LIN {X 0,Y 239.969,Z 223.755,A -85,B 0,C 180,E1 -22346.527,E2 -22346.527} C_VEL
LIN {X 0,Y 242.861,Z 228.839,A -85,B 0,C 180,E1 -22348.912,E2 -22348.912} C_VEL
LIN {X 0,Y 246.024,Z 234.682,A -85,B 0,C 180,E1 -22351.164,E2 -22351.164} C_VEL
LIN {X 0,Y 248.847,Z 240.046,A -85,B 0,C 180,E1 -22352.983,E2 -22352.983} C_VEL
LIN {X 0,Y 253.177,Z 249.294,A -85,B 0,C 180,E1 -22355.55,E2 -22355.55} C_VEL
LIN {X 0,Y 256.52,Z 257.154,A -85,B 0,C 180,E1 -22357.368,E2 -22357.368} C_VEL
LIN {X 0,Y 257.027,Z 259.364,A -85,B 0,C 180,E1 -22357.681,E2 -22357.681} C_VEL
LIN {X 0,Y 256.983,Z 262.913,A -85,B 0,C 180,E1 -22357.859,E2 -22357.859} C_VEL
LIN {X 0,Y 256.14,Z 267.671,A -85,B 0,C 180,E1 -22357.804,E2 -22357.804} C_VEL
LIN {X 0,Y 255.103,Z 271.378,A -85,B 0,C 180,E1 -22357.618,E2 -22357.618} C_VEL
LIN {X 0,Y 251.834,Z 281.658,A -85,B 0,C 180,E1 -22356.935,E2 -22356.935} C_VEL
LIN {X 0,Y 250.756,Z 287.02,A -85,B 0,C 180,E1 -22356.819,E2 -22356.819} C_VEL
LIN {X 0,Y 250.638,Z 288.109,A -85,B 0,C 180,E1 -22356.836,E2 -22356.836} C_VEL
LIN {X 0,Y 247.434,Z 325.09,A -85,B 0,C 180,E1 -22357.818,E2 -22357.818} C_VEL
LIN {X 0,Y 244.93,Z 340.568,A -85,B 0,C 180,E1 -22358.4,E2 -22358.4} C_VEL
LIN {X 0,Y 241.457,Z 355.534,A -85,B 0,C 180,E1 -22359.199,E2 -22359.199} C_VEL
LIN {X 0,Y 237.664,Z 368.105,A -85,B 0,C 180,E1 -22360.08,E2 -22360.08} C_VEL
LIN {X 0,Y 232.84,Z 381.625,A -85,B 0,C 180,E1 -22361.339,E2 -22361.339} C_VEL
LIN {X 0,Y 227.303,Z 394.667,A -85,B 0,C 180,E1 -22362.894,E2 -22362.894} C_VEL
LIN {X 0,Y 221.538,Z 406.76,A -85,B 0,C 180,E1 -22364.781,E2 -22364.781} C_VEL
LIN {X 0,Y 216.696,Z 415.667,A -85,B 0,C 180,E1 -22366.435,E2 -22366.435} C_VEL
LIN {X 0,Y 210.539,Z 425.809,A -85,B 0,C 180,E1 -22368.756,E2 -22368.756} C_VEL
LIN {X 0,Y 203.927,Z 435.781,A -85,B 0,C 180,E1 -22371.66,E2 -22371.66} C_VEL
LIN {X 0,Y 197.461,Z 444.613,A -85,B 0,C 180,E1 -22374.945,E2 -22374.945} C_VEL
LIN {X 0,Y 192.716,Z 451.07,A -85,B 0,C 180,E1 -22378.077,E2 -22378.077} C_VEL
LIN {X 0,Y 187.417,Z 457.586,A -85,B 0,C 180,E1 -22382.048,E2 -22382.048} C_VEL
LIN {X 0,Y 183.132,Z 462.73,A -85,B 0,C 180,E1 -22386.238,E2 -22386.238} C_VEL
LIN {X 0,Y 180.543,Z 465.734,A -85,B 0,C 180,E1 -22389.493,E2 -22389.493} C_VEL
LIN {X 0,Y 178.115,Z 468.722,A -85,B 0,C 180,E1 -22393.967,E2 -22393.967} C_VEL
LIN {X 0,Y 176.609,Z 470.59,A -85,B 0,C 180,E1 -22398.524,E2 -22398.524} C_VEL
LIN {X 0,Y 175.965,Z 471.317,A -85,B 0,C 180,E1 -22403.119,E2 -22403.119} C_VEL
LIN {X 0,Y 175.967,Z 470.901,A -85,B 0,C 180,E1 -22407.712,E2 -22407.712} C_VEL
LIN {X 0,Y 176.119,Z 470.269,A -85,B 0,C 180,E1 -22410.001,E2 -22410.001} C_VEL
LIN {X 0,Y 176.018,Z 468.093,A -85,B 0,C 180,E1 -22414.581,E2 -22414.581} C_VEL
LIN {X 0,Y 176.233,Z 464.666,A -85,B 0,C 180,E1 -22419.18,E2 -22419.18} C_VEL
LIN {X 0,Y 177.037,Z 459.891,A -85,B 0,C 180,E1 -22423.781,E2 -22423.781} C_VEL
LIN {X 0,Y 178.755,Z 453.644,A -85,B 0,C 180,E1 -22428.334,E2 -22428.334} C_VEL
LIN {X 0,Y 181.359,Z 445.739,A -85,B 0,C 180,E1 -22432.801,E2 -22432.801} C_VEL
LIN {X 0,Y 184.466,Z 437.297,A -85,B 0,C 180,E1 -22436.595,E2 -22436.595} C_VEL
LIN {X 0,Y 188.286,Z 427.088,A -85,B 0,C 180,E1 -22440.26,E2 -22440.26} C_VEL
LIN {X 0,Y 192.055,Z 416.618,A -85,B 0,C 180,E1 -22443.293,E2 -22443.293} C_VEL
LIN {X 0,Y 196.36,Z 404.072,A -85,B 0,C 180,E1 -22446.198,E2 -22446.198} C_VEL
LIN {X 0,Y 199.968,Z 392.825,A -85,B 0,C 180,E1 -22448.277,E2 -22448.277} C_VEL
LIN {X 0,Y 203.401,Z 380.951,A -85,B 0,C 180,E1 -22450.057,E2 -22450.057} C_VEL
LIN {X 0,Y 206.679,Z 367.637,A -85,B 0,C 180,E1 -22451.668,E2 -22451.668} C_VEL
LIN {X 0,Y 209.533,Z 353.912,A -85,B 0,C 180,E1 -22452.947,E2 -22452.947} C_VEL
LIN {X 0,Y 211.958,Z 339.018,A -85,B 0,C 180,E1 -22453.968,E2 -22453.968} C_VEL
LIN {X 0,Y 213.625,Z 323.778,A -85,B 0,C 180,E1 -22454.686,E2 -22454.686} C_VEL
LIN {X 0,Y 218.933,Z 239.212,A -85,B 0,C 180,E1 -22457.242,E2 -22457.242} C_VEL
LIN {X 0,Y 218.792,Z 237.497,A -85,B 0,C 180,E1 -22457.347,E2 -22457.347} C_VEL
LIN {X 0,Y 212.348,Z 220.9,A -85,B 0,C 180,E1 -22459.583,E2 -22459.583} C_VEL
LIN {X 0,Y 206.415,Z 207.779,A -85,B 0,C 180,E1 -22461.739,E2 -22461.739} C_VEL
LIN {X 0,Y 200.574,Z 196.158,A -85,B 0,C 180,E1 -22464.009,E2 -22464.009} C_VEL
LIN {X 0,Y 196.878,Z 189.859,A -85,B 0,C 180,E1 -22465.51,E2 -22465.51} C_VEL
LIN {X 0,Y 191.655,Z 182.342,A -85,B 0,C 180,E1 -22467.702,E2 -22467.702} C_VEL
LIN {X 0,Y 188.625,Z 178.111,A -85,B 0,C 180,E1 -22469.066,E2 -22469.066} C_VEL
LIN {X 0,Y 185.755,Z 174.12,A -85,B 0,C 180,E1 -22470.429,E2 -22470.429} C_VEL
LIN {X 0,Y 183.259,Z 171.243,A -85,B 0,C 180,E1 -22471.647,E2 -22471.647} C_VEL
LIN {X 0,Y 182.122,Z 169.152,A -85,B 0,C 180,E1 -22472.278,E2 -22472.278} C_VEL
LIN {X 0,Y 179.819,Z 167.216,A -85,B 0,C 180,E1 -22473.448,E2 -22473.448} C_VEL
LIN {X 0,Y 178.609,Z 164.655,A -85,B 0,C 180,E1 -22474.197,E2 -22474.197} C_VEL
LIN {X 0,Y 178.489,Z 163.848,A -85,B 0,C 180,E1 -22474.335,E2 -22474.335} C_VEL
LIN {X 0,Y 178.521,Z 163.862,A -85,B 0,C 180,E1 -22479.25,E2 -22479.25} C_VEL
LIN {X 0,Y 178.649,Z 163.849,A -85,B 0,C 180,E1 -22481.657,E2 -22481.657} C_VEL
LIN {X 0,Y 178.653,Z 163.852,A -85,B 0,C 180,E1 -22486.348,E2 -22486.348} C_VEL
LIN {X 0,Y 178.908,Z 163.82,A -85,B 0,C 180,E1 -22490.961,E2 -22490.961} C_VEL
LIN {X 0,Y 179.128,Z 163.756,A -85,B 0,C 180,E1 -22497.752,E2 -22497.752} C_VEL
LIN {X 0,Y 179.348,Z 163.718,A -85,B 0,C 180,E1 -22500.001,E2 -22500.001} C_VEL
LIN {X 0,Y 178.834,Z 163.832,A -85,B 0,C 180,E1 -22504.509,E2 -22504.509} C_VEL
LIN {X 0,Y 178.907,Z 163.771,A -85,B 0,C 180,E1 -22509.041,E2 -22509.041} C_VEL
LIN {X 0,Y 178.633,Z 163.853,A -85,B 0,C 180,E1 -22513.655,E2 -22513.655} C_VEL
LIN {X 0,Y 178.558,Z 163.866,A -85,B 0,C 180,E1 -22519.151,E2 -22519.151} C_VEL
LIN {X 0,Y 178.509,Z 163.873,A -85,B 0,C 180,E1 -22525.104,E2 -22525.104} C_VEL
LIN {X 0,Y 178.465,Z 163.836,A -85,B 0,C 180,E1 -22530.795,E2 -22530.795} C_VEL
LIN {X 0,Y 178.487,Z 163.876,A -85,B 0,C 180,E1 -22534.218,E2 -22534.218} C_VEL
LIN {X 0,Y 178.392,Z 163.849,A -85,B 0,C 180,E1 -22539.077,E2 -22539.077} C_VEL
LIN {X 0,Y 178.399,Z 163.887,A -85,B 0,C 180,E1 -22542.046,E2 -22542.046} C_VEL
LIN {X 0,Y 178.436,Z 164.055,A -85,B 0,C 180,E1 -22545.152,E2 -22545.152} C_VEL
LIN {X 0,Y 179.226,Z 166.376,A -85,B 0,C 180,E1 -22545.697,E2 -22545.697} C_VEL
LIN {X 0,Y 181.252,Z 168.699,A -85,B 0,C 180,E1 -22546.789,E2 -22546.789} C_VEL
LIN {X 0,Y 182.292,Z 169.507,A -85,B 0,C 180,E1 -22547.302,E2 -22547.302} C_VEL
LIN {X 0,Y 184.39,Z 172.908,A -85,B 0,C 180,E1 -22548.419,E2 -22548.419} C_VEL
LIN {X 0,Y 186.241,Z 174.918,A -85,B 0,C 180,E1 -22549.298,E2 -22549.298} C_VEL
LIN {X 0,Y 188.955,Z 178.567,A -85,B 0,C 180,E1 -22550.569,E2 -22550.569} C_VEL
LIN {X 0,Y 195.455,Z 187.623,A -85,B 0,C 180,E1 -22553.375,E2 -22553.375} C_VEL
LIN {X 0,Y 203.125,Z 199.683,A -85,B 0,C 180,E1 -22556.407,E2 -22556.407} C_VEL
LIN {X 0,Y 210.617,Z 212.759,A -85,B 0,C 180,E1 -22559.08,E2 -22559.08} C_VEL
LIN {X 0,Y 216.744,Z 224.617,A -85,B 0,C 180,E1 -22561.105,E2 -22561.105} C_VEL
LIN {X 0,Y 219.28,Z 230.916,A -85,B 0,C 180,E1 -22561.953,E2 -22561.953} C_VEL
LIN {X 0,Y 213.746,Z 316.637,A -85,B 0,C 180,E1 -22564.531,E2 -22564.531} C_VEL
LIN {X 0,Y 211.892,Z 332.826,A -85,B 0,C 180,E1 -22565.374,E2 -22565.374} C_VEL
LIN {X 0,Y 209.446,Z 347.863,A -85,B 0,C 180,E1 -22566.517,E2 -22566.517} C_VEL
LIN {X 0,Y 206.413,Z 362.396,A -85,B 0,C 180,E1 -22568.004,E2 -22568.004} C_VEL
LIN {X 0,Y 202.845,Z 376.704,A -85,B 0,C 180,E1 -22569.919,E2 -22569.919} C_VEL
LIN {X 0,Y 199.173,Z 389.206,A -85,B 0,C 180,E1 -22572.015,E2 -22572.015} C_VEL
LIN {X 0,Y 195.103,Z 401.514,A -85,B 0,C 180,E1 -22574.593,E2 -22574.593} C_VEL
LIN {X 0,Y 191.448,Z 411.856,A -85,B 0,C 180,E1 -22577.275,E2 -22577.275} C_VEL
LIN {X 0,Y 187.329,Z 422.924,A -85,B 0,C 180,E1 -22580.824,E2 -22580.824} C_VEL
LIN {X 0,Y 183.74,Z 432.584,A -85,B 0,C 180,E1 -22584.751,E2 -22584.751} C_VEL
LIN {X 0,Y 180.767,Z 440.674,A -85,B 0,C 180,E1 -22588.885,E2 -22588.885} C_VEL
LIN {X 0,Y 178.476,Z 447.58,A -85,B 0,C 180,E1 -22593.385,E2 -22593.385} C_VEL
LIN {X 0,Y 177.118,Z 452.205,A -85,B 0,C 180,E1 -22597.246,E2 -22597.246} C_VEL
LIN {X 0,Y 176.116,Z 456.146,A -85,B 0,C 180,E1 -22601.508,E2 -22601.508} C_VEL
LIN {X 0,Y 175.623,Z 459.251,A -85,B 0,C 180,E1 -22606.267,E2 -22606.267} C_VEL
LIN {X 0,Y 175.616,Z 461.112,A -85,B 0,C 180,E1 -22611.11,E2 -22611.11} C_VEL
LIN {X 0,Y 175.839,Z 461.573,A -85,B 0,C 180,E1 -22613.557,E2 -22613.557} C_VEL
LIN {X 0,Y 176.766,Z 461.54,A -85,B 0,C 180,E1 -22618.496,E2 -22618.496} C_VEL
LIN {X 0,Y 178.583,Z 460.199,A -85,B 0,C 180,E1 -22623.432,E2 -22623.432} C_VEL
LIN {X 0,Y 181.425,Z 457.485,A -85,B 0,C 180,E1 -22628.301,E2 -22628.301} C_VEL
LIN {X 0,Y 185.362,Z 453.318,A -85,B 0,C 180,E1 -22633.036,E2 -22633.036} C_VEL
LIN {X 0,Y 190.406,Z 447.573,A -85,B 0,C 180,E1 -22637.578,E2 -22637.578} C_VEL
LIN {X 0,Y 195.755,Z 441.141,A -85,B 0,C 180,E1 -22641.339,E2 -22641.339} C_VEL
LIN {X 0,Y 201.83,Z 433.164,A -85,B 0,C 180,E1 -22644.914,E2 -22644.914} C_VEL
LIN {X 0,Y 208.702,Z 423.409,A -85,B 0,C 180,E1 -22648.242,E2 -22648.242} C_VEL
LIN {X 0,Y 214.787,Z 413.801,A -85,B 0,C 180,E1 -22650.814,E2 -22650.814} C_VEL
LIN {X 0,Y 220.727,Z 403.292,A -85,B 0,C 180,E1 -22653.064,E2 -22653.064} C_VEL
LIN {X 0,Y 226.688,Z 391.48,A -85,B 0,C 180,E1 -22655.071,E2 -22655.071} C_VEL
LIN {X 0,Y 232.35,Z 378.396,A -85,B 0,C 180,E1 -22656.844,E2 -22656.844} C_VEL
LIN {X 0,Y 236.716,Z 366.66,A -85,B 0,C 180,E1 -22658.093,E2 -22658.093} C_VEL
LIN {X 0,Y 241.007,Z 352.669,A -85,B 0,C 180,E1 -22659.279,E2 -22659.279} C_VEL
LIN {X 0,Y 244.365,Z 338.95,A -85,B 0,C 180,E1 -22660.163,E2 -22660.163} C_VEL
LIN {X 0,Y 247.197,Z 323.376,A -85,B 0,C 180,E1 -22660.868,E2 -22660.868} C_VEL
LIN {X 0,Y 249.061,Z 306.485,A -85,B 0,C 180,E1 -22661.377,E2 -22661.377} C_VEL
LIN {X 0,Y 253.376,Z 254.975,A -85,B 0,C 180,E1 -22662.68,E2 -22662.68} C_VEL
LIN {X 0,Y 250.863,Z 249.621,A -85,B 0,C 180,E1 -22664.101,E2 -22664.101} C_VEL
LIN {X 0,Y 246.36,Z 241.669,A -85,B 0,C 180,E1 -22666.807,E2 -22666.807} C_VEL
LIN {X 0,Y 242.061,Z 234.701,A -85,B 0,C 180,E1 -22669.746,E2 -22669.746} C_VEL
LIN {X 0,Y 239.686,Z 230.917,A -85,B 0,C 180,E1 -22671.655,E2 -22671.655} C_VEL
LIN {X 0,Y 236.901,Z 226.565,A -85,B 0,C 180,E1 -22674.234,E2 -22674.234} C_VEL
LIN {X 0,Y 234.776,Z 223.186,A -85,B 0,C 180,E1 -22676.567,E2 -22676.567} C_VEL
LIN {X 0,Y 232.594,Z 220.661,A -85,B 0,C 180,E1 -22679.373,E2 -22679.373} C_VEL
LIN {X 0,Y 231.552,Z 218.244,A -85,B 0,C 180,E1 -22681.402,E2 -22681.402} C_VEL
LIN {X 0,Y 229.408,Z 216.365,A -85,B 0,C 180,E1 -22688.81,E2 -22688.81} C_VEL
LIN {X 0,Y 230.648,Z 217.994,A -85,B 0,C 180,E1 -22695.473,E2 -22695.473} C_VEL
LIN {X 0,Y 231.612,Z 218.858,A -85,B 0,C 180,E1 -22697.498,E2 -22697.498} C_VEL
LIN {X 0,Y 233.569,Z 222.339,A -85,B 0,C 180,E1 -22700.708,E2 -22700.708} C_VEL
LIN {X 0,Y 235.227,Z 224.477,A -85,B 0,C 180,E1 -22702.696,E2 -22702.696} C_VEL
LIN {X 0,Y 238.452,Z 230.475,A -85,B 0,C 180,E1 -22706.066,E2 -22706.066} C_VEL
LIN {X 0,Y 240.896,Z 234.97,A -85,B 0,C 180,E1 -22708.203,E2 -22708.203} C_VEL
LIN {X 0,Y 244.031,Z 240.978,A -85,B 0,C 180,E1 -22710.552,E2 -22710.552} C_VEL
LIN {X 0,Y 247.014,Z 247.044,A -85,B 0,C 180,E1 -22712.564,E2 -22712.564} C_VEL
LIN {X 0,Y 251.252,Z 256.485,A -85,B 0,C 180,E1 -22715.165,E2 -22715.165} C_VEL
LIN {X 0,Y 252.923,Z 260.745,A -85,B 0,C 180,E1 -22716.14,E2 -22716.14} C_VEL
LIN {X 0,Y 250.638,Z 288.109,A -85,B 0,C 180,E1 -22716.836,E2 -22716.836} C_VEL
LIN {X 0,Y 249.82,Z 293.964,A -85,B 0,C 180,E1 -22716.842,E2 -22716.842} C_VEL
LIN {X 0,Y 245.488,Z 313.103,A -85,B 0,C 180,E1 -22716.176,E2 -22716.176} C_VEL
LIN {X 0,Y 244.576,Z 318.943,A -85,B 0,C 180,E1 -22716.193,E2 -22716.193} C_VEL
LIN {X 0,Y 242.481,Z 334.567,A -85,B 0,C 180,E1 -22716.72,E2 -22716.72} C_VEL
LIN {X 0,Y 239.327,Z 349.266,A -85,B 0,C 180,E1 -22717.373,E2 -22717.373} C_VEL
LIN {X 0,Y 235.757,Z 362.161,A -85,B 0,C 180,E1 -22718.165,E2 -22718.165} C_VEL
LIN {X 0,Y 230.748,Z 376.824,A -85,B 0,C 180,E1 -22719.39,E2 -22719.39} C_VEL
LIN {X 0,Y 224.657,Z 391.382,A -85,B 0,C 180,E1 -22721.001,E2 -22721.001} C_VEL
LIN {X 0,Y 219.383,Z 402.272,A -85,B 0,C 180,E1 -22722.54,E2 -22722.54} C_VEL
LIN {X 0,Y 212.739,Z 414.522,A -85,B 0,C 180,E1 -22724.744,E2 -22724.744} C_VEL
LIN {X 0,Y 205.283,Z 426.409,A -85,B 0,C 180,E1 -22727.457,E2 -22727.457} C_VEL
LIN {X 0,Y 198.412,Z 436.254,A -85,B 0,C 180,E1 -22730.389,E2 -22730.389} C_VEL
LIN {X 0,Y 191.234,Z 445.554,A -85,B 0,C 180,E1 -22733.985,E2 -22733.985} C_VEL
LIN {X 0,Y 185.216,Z 453.106,A -85,B 0,C 180,E1 -22737.912,E2 -22737.912} C_VEL
LIN {X 0,Y 179.938,Z 459.164,A -85,B 0,C 180,E1 -22742.051,E2 -22742.051} C_VEL
LIN {X 0,Y 175.643,Z 463.869,A -85,B 0,C 180,E1 -22746.415,E2 -22746.415} C_VEL
LIN {X 0,Y 172.428,Z 467.353,A -85,B 0,C 180,E1 -22750.97,E2 -22750.97} C_VEL
LIN {X 0,Y 170.272,Z 469.692,A -85,B 0,C 180,E1 -22755.662,E2 -22755.662} C_VEL
LIN {X 0,Y 169.159,Z 470.933,A -85,B 0,C 180,E1 -22760.435,E2 -22760.435} C_VEL
LIN {X 0,Y 168.793,Z 471.029,A -85,B 0,C 180,E1 -22765.224,E2 -22765.224} C_VEL
LIN {X 0,Y 169.025,Z 469.979,A -85,B 0,C 180,E1 -22770.001,E2 -22770.001} C_VEL
LIN {X 0,Y 168.929,Z 467.728,A -85,B 0,C 180,E1 -22774.774,E2 -22774.774} C_VEL
LIN {X 0,Y 169.169,Z 464.221,A -85,B 0,C 180,E1 -22779.567,E2 -22779.567} C_VEL
LIN {X 0,Y 170.083,Z 459.363,A -85,B 0,C 180,E1 -22784.356,E2 -22784.356} C_VEL
LIN {X 0,Y 171.929,Z 453.023,A -85,B 0,C 180,E1 -22789.089,E2 -22789.089} C_VEL
LIN {X 0,Y 174.741,Z 445.012,A -85,B 0,C 180,E1 -22793.717,E2 -22793.717} C_VEL
LIN {X 0,Y 178.081,Z 436.456,A -85,B 0,C 180,E1 -22797.628,E2 -22797.628} C_VEL
LIN {X 0,Y 181.455,Z 427.767,A -85,B 0,C 180,E1 -22800.86,E2 -22800.86} C_VEL
LIN {X 0,Y 185.684,Z 416.547,A -85,B 0,C 180,E1 -22804.232,E2 -22804.232} C_VEL
LIN {X 0,Y 189.797,Z 405.03,A -85,B 0,C 180,E1 -22806.995,E2 -22806.995} C_VEL
LIN {X 0,Y 193.516,Z 393.964,A -85,B 0,C 180,E1 -22809.126,E2 -22809.126} C_VEL
LIN {X 0,Y 197.014,Z 382.366,A -85,B 0,C 180,E1 -22810.958,E2 -22810.958} C_VEL
LIN {X 0,Y 200.724,Z 368.114,A -85,B 0,C 180,E1 -22812.741,E2 -22812.741} C_VEL
LIN {X 0,Y 203.571,Z 354.999,A -85,B 0,C 180,E1 -22814.011,E2 -22814.011} C_VEL
LIN {X 0,Y 206.199,Z 339.703,A -85,B 0,C 180,E1 -22815.098,E2 -22815.098} C_VEL
LIN {X 0,Y 207.952,Z 325.05,A -85,B 0,C 180,E1 -22815.818,E2 -22815.818} C_VEL
LIN {X 0,Y 213.471,Z 240.252,A -85,B 0,C 180,E1 -22818.43,E2 -22818.43} C_VEL
LIN {X 0,Y 208.078,Z 225.803,A -85,B 0,C 180,E1 -22820.424,E2 -22820.424} C_VEL
LIN {X 0,Y 202.206,Z 212.376,A -85,B 0,C 180,E1 -22822.683,E2 -22822.683} C_VEL
LIN {X 0,Y 196.177,Z 200.155,A -85,B 0,C 180,E1 -22825.164,E2 -22825.164} C_VEL
LIN {X 0,Y 192.962,Z 194.707,A -85,B 0,C 180,E1 -22826.535,E2 -22826.535} C_VEL
LIN {X 0,Y 187.957,Z 187.439,A -85,B 0,C 180,E1 -22828.741,E2 -22828.741} C_VEL
LIN {X 0,Y 184.763,Z 182.963,A -85,B 0,C 180,E1 -22830.255,E2 -22830.255} C_VEL
LIN {X 0,Y 182.514,Z 179.81,A -85,B 0,C 180,E1 -22831.386,E2 -22831.386} C_VEL
LIN {X 0,Y 179.904,Z 176.41,A -85,B 0,C 180,E1 -22832.756,E2 -22832.756} C_VEL
LIN {X 0,Y 179.148,Z 175.224,A -85,B 0,C 180,E1 -22833.184,E2 -22833.184} C_VEL
LIN {X 0,Y 176.649,Z 172.6,A -85,B 0,C 180,E1 -22834.558,E2 -22834.558} C_VEL
LIN {X 0,Y 175.347,Z 170.224,A -85,B 0,C 180,E1 -22835.384,E2 -22835.384} C_VEL
LIN {X 0,Y 173.019,Z 168.352,A -85,B 0,C 180,E1 -22836.749,E2 -22836.749} C_VEL
LIN {X 0,Y 171.78,Z 166.247,A -85,B 0,C 180,E1 -22837.605,E2 -22837.605} C_VEL
LIN {X 0,Y 171.448,Z 164.74,A -85,B 0,C 180,E1 -22838.035,E2 -22838.035} C_VEL
LIN {X 0,Y 171.579,Z 164.736,A -85,B 0,C 180,E1 -22840.873,E2 -22840.873} C_VEL
LIN {X 0,Y 171.571,Z 164.739,A -85,B 0,C 180,E1 -22845.773,E2 -22845.773} C_VEL
LIN {X 0,Y 171.847,Z 164.702,A -85,B 0,C 180,E1 -22850.586,E2 -22850.586} C_VEL
LIN {X 0,Y 171.789,Z 164.709,A -85,B 0,C 180,E1 -22855.308,E2 -22855.308} C_VEL
LIN {X 0,Y 172.313,Z 164.594,A -85,B 0,C 180,E1 -22860.001,E2 -22860.001} C_VEL
LIN {X 0,Y 171.784,Z 164.71,A -85,B 0,C 180,E1 -22864.694,E2 -22864.694} C_VEL
LIN {X 0,Y 171.846,Z 164.649,A -85,B 0,C 180,E1 -22869.416,E2 -22869.416} C_VEL
LIN {X 0,Y 171.547,Z 164.74,A -85,B 0,C 180,E1 -22874.231,E2 -22874.231} C_VEL
LIN {X 0,Y 171.483,Z 164.749,A -85,B 0,C 180,E1 -22879.499,E2 -22879.499} C_VEL
LIN {X 0,Y 171.439,Z 164.749,A -85,B 0,C 180,E1 -22885.592,E2 -22885.592} C_VEL
LIN {X 0,Y 171.422,Z 164.711,A -85,B 0,C 180,E1 -22890.573,E2 -22890.573} C_VEL
LIN {X 0,Y 171.396,Z 164.75,A -85,B 0,C 180,E1 -22895.035,E2 -22895.035} C_VEL
LIN {X 0,Y 171.348,Z 164.724,A -85,B 0,C 180,E1 -22898.801,E2 -22898.801} C_VEL
LIN {X 0,Y 171.377,Z 164.899,A -85,B 0,C 180,E1 -22901.53,E2 -22901.53} C_VEL
LIN {X 0,Y 172.392,Z 167.7,A -85,B 0,C 180,E1 -22902.328,E2 -22902.328} C_VEL
LIN {X 0,Y 174.376,Z 169.75,A -85,B 0,C 180,E1 -22903.549,E2 -22903.549} C_VEL
LIN {X 0,Y 175.546,Z 170.593,A -85,B 0,C 180,E1 -22904.217,E2 -22904.217} C_VEL
LIN {X 0,Y 177.542,Z 173.816,A -85,B 0,C 180,E1 -22905.443,E2 -22905.443} C_VEL
LIN {X 0,Y 179.575,Z 175.952,A -85,B 0,C 180,E1 -22906.544,E2 -22906.544} C_VEL
LIN {X 0,Y 182.078,Z 179.473,A -85,B 0,C 180,E1 -22907.888,E2 -22907.888} C_VEL
LIN {X 0,Y 183.467,Z 181.249,A -85,B 0,C 180,E1 -22908.589,E2 -22908.589} C_VEL
LIN {X 0,Y 187.359,Z 186.619,A -85,B 0,C 180,E1 -22910.467,E2 -22910.467} C_VEL
LIN {X 0,Y 192.425,Z 193.854,A -85,B 0,C 180,E1 -22912.712,E2 -22912.712} C_VEL
LIN {X 0,Y 200.132,Z 206.208,A -85,B 0,C 180,E1 -22915.865,E2 -22915.865} C_VEL
LIN {X 0,Y 207.853,Z 220.313,A -85,B 0,C 180,E1 -22918.729,E2 -22918.729} C_VEL
LIN {X 0,Y 213.062,Z 230.924,A -85,B 0,C 180,E1 -22920.526,E2 -22920.526} C_VEL
LIN {X 0,Y 213.739,Z 232.552,A -85,B 0,C 180,E1 -22920.76,E2 -22920.76} C_VEL
LIN {X 0,Y 208.137,Z 317.01,A -85,B 0,C 180,E1 -22923.354,E2 -22923.354} C_VEL
LIN {X 0,Y 206.279,Z 332.759,A -85,B 0,C 180,E1 -22924.184,E2 -22924.184} C_VEL
LIN {X 0,Y 203.855,Z 347.296,A -85,B 0,C 180,E1 -22925.29,E2 -22925.29} C_VEL
LIN {X 0,Y 200.712,Z 361.995,A -85,B 0,C 180,E1 -22926.8,E2 -22926.8} C_VEL
LIN {X 0,Y 197.3,Z 375.358,A -85,B 0,C 180,E1 -22928.584,E2 -22928.584} C_VEL
LIN {X 0,Y 193.178,Z 389.007,A -85,B 0,C 180,E1 -22930.886,E2 -22930.886} C_VEL
LIN {X 0,Y 188.972,Z 401.383,A -85,B 0,C 180,E1 -22933.525,E2 -22933.525} C_VEL
LIN {X 0,Y 184.51,Z 413.487,A -85,B 0,C 180,E1 -22936.788,E2 -22936.788} C_VEL
LIN {X 0,Y 180.835,Z 422.9,A -85,B 0,C 180,E1 -22939.927,E2 -22939.927} C_VEL
LIN {X 0,Y 177.307,Z 432.027,A -85,B 0,C 180,E1 -22943.713,E2 -22943.713} C_VEL
LIN {X 0,Y 174.29,Z 439.734,A -85,B 0,C 180,E1 -22947.688,E2 -22947.688} C_VEL
LIN {X 0,Y 171.735,Z 446.882,A -85,B 0,C 180,E1 -22952.344,E2 -22952.344} C_VEL
LIN {X 0,Y 170.008,Z 452.559,A -85,B 0,C 180,E1 -22957.177,E2 -22957.177} C_VEL
LIN {X 0,Y 168.919,Z 456.75,A -85,B 0,C 180,E1 -22962.006,E2 -22962.006} C_VEL
LIN {X 0,Y 168.463,Z 459.713,A -85,B 0,C 180,E1 -22966.979,E2 -22966.979} C_VEL
LIN {X 0,Y 168.575,Z 461.43,A -85,B 0,C 180,E1 -22972.037,E2 -22972.037} C_VEL
LIN {X 0,Y 168.843,Z 461.822,A -85,B 0,C 180,E1 -22974.597,E2 -22974.597} C_VEL
LIN {X 0,Y 169.986,Z 461.645,A -85,B 0,C 180,E1 -22979.744,E2 -22979.744} C_VEL
LIN {X 0,Y 172.103,Z 460.156,A -85,B 0,C 180,E1 -22984.868,E2 -22984.868} C_VEL
LIN {X 0,Y 175.343,Z 457.293,A -85,B 0,C 180,E1 -22989.888,E2 -22989.888} C_VEL
LIN {X 0,Y 179.676,Z 452.961,A -85,B 0,C 180,E1 -22994.753,E2 -22994.753} C_VEL
LIN {X 0,Y 185.209,Z 447.044,A -85,B 0,C 180,E1 -22999.369,E2 -22999.369} C_VEL
LIN {X 0,Y 190.919,Z 440.431,A -85,B 0,C 180,E1 -23003.191,E2 -23003.191} C_VEL
LIN {X 0,Y 197.425,Z 432.257,A -85,B 0,C 180,E1 -23006.778,E2 -23006.778} C_VEL
LIN {X 0,Y 203.622,Z 423.851,A -85,B 0,C 180,E1 -23009.639,E2 -23009.639} C_VEL
LIN {X 0,Y 210.599,Z 413.217,A -85,B 0,C 180,E1 -23012.487,E2 -23012.487} C_VEL
LIN {X 0,Y 216.721,Z 402.773,A -85,B 0,C 180,E1 -23014.681,E2 -23014.681} C_VEL
LIN {X 0,Y 222.905,Z 390.831,A -85,B 0,C 180,E1 -23016.675,E2 -23016.675} C_VEL
LIN {X 0,Y 228.43,Z 378.427,A -85,B 0,C 180,E1 -23018.333,E2 -23018.333} C_VEL
LIN {X 0,Y 233.264,Z 365.674,A -85,B 0,C 180,E1 -23019.678,E2 -23019.678} C_VEL
LIN {X 0,Y 237.78,Z 351.178,A -85,B 0,C 180,E1 -23020.858,E2 -23020.858} C_VEL
LIN {X 0,Y 241.065,Z 337.796,A -85,B 0,C 180,E1 -23021.678,E2 -23021.678} C_VEL
LIN {X 0,Y 243.892,Z 322.153,A -85,B 0,C 180,E1 -23022.354,E2 -23022.354} C_VEL
LIN {X 0,Y 245.801,Z 304.505,A -85,B 0,C 180,E1 -23022.861,E2 -23022.861} C_VEL
LIN {X 0,Y 249.753,Z 258.274,A -85,B 0,C 180,E1 -23024.045,E2 -23024.045} C_VEL
LIN {X 0,Y 246.634,Z 252.054,A -85,B 0,C 180,E1 -23025.933,E2 -23025.933} C_VEL
LIN {X 0,Y 242.062,Z 244.117,A -85,B 0,C 180,E1 -23028.978,E2 -23028.978} C_VEL
LIN {X 0,Y 238.436,Z 237.966,A -85,B 0,C 180,E1 -23031.871,E2 -23031.871} C_VEL
LIN {X 0,Y 235.316,Z 233.038,A -85,B 0,C 180,E1 -23034.859,E2 -23034.859} C_VEL
LIN {X 0,Y 233.397,Z 229.945,A -85,B 0,C 180,E1 -23037.074,E2 -23037.074} C_VEL
LIN {X 0,Y 231.247,Z 227.111,A -85,B 0,C 180,E1 -23040.094,E2 -23040.094} C_VEL
LIN {X 0,Y 230.469,Z 225.176,A -85,B 0,C 180,E1 -23041.747,E2 -23041.747} C_VEL
LIN {X 0,Y 228.511,Z 223.414,A -85,B 0,C 180,E1 -23048.845,E2 -23048.845} C_VEL
LIN {X 0,Y 229.778,Z 225.052,A -85,B 0,C 180,E1 -23055.533,E2 -23055.533} C_VEL
LIN {X 0,Y 230.525,Z 225.778,A -85,B 0,C 180,E1 -23057.154,E2 -23057.154} C_VEL
LIN {X 0,Y 232.536,Z 229.359,A -85,B 0,C 180,E1 -23060.567,E2 -23060.567} C_VEL
LIN {X 0,Y 233.903,Z 231.317,A -85,B 0,C 180,E1 -23062.276,E2 -23062.276} C_VEL
LIN {X 0,Y 236.798,Z 236.909,A -85,B 0,C 180,E1 -23065.454,E2 -23065.454} C_VEL
LIN {X 0,Y 238.972,Z 241.013,A -85,B 0,C 180,E1 -23067.456,E2 -23067.456} C_VEL
LIN {X 0,Y 242.914,Z 248.905,A -85,B 0,C 180,E1 -23070.54,E2 -23070.54} C_VEL
LIN {X 0,Y 247.345,Z 258.987,A -85,B 0,C 180,E1 -23073.545,E2 -23073.545} C_VEL
LIN {X 0,Y 249.32,Z 263.896,A -85,B 0,C 180,E1 -23074.779,E2 -23074.779} C_VEL
LIN {X 0,Y 244.576,Z 318.943,A -85,B 0,C 180,E1 -23076.193,E2 -23076.193} C_VEL
LIN {X 0,Y 243.597,Z 324.771,A -85,B 0,C 180,E1 -23076.208,E2 -23076.208} C_VEL
LIN {X 0,Y 240.799,Z 334.234,A -85,B 0,C 180,E1 -23075.953,E2 -23075.953} C_VEL
LIN {X 0,Y 237.583,Z 343.569,A -85,B 0,C 180,E1 -23075.745,E2 -23075.745} C_VEL
LIN {X 0,Y 235.861,Z 349.193,A -85,B 0,C 180,E1 -23075.877,E2 -23075.877} C_VEL
LIN {X 0,Y 232.177,Z 362.162,A -85,B 0,C 180,E1 -23076.664,E2 -23076.664} C_VEL
LIN {X 0,Y 227.015,Z 376.784,A -85,B 0,C 180,E1 -23077.868,E2 -23077.868} C_VEL
LIN {X 0,Y 221.388,Z 390.014,A -85,B 0,C 180,E1 -23079.306,E2 -23079.306} C_VEL
LIN {X 0,Y 215.69,Z 401.388,A -85,B 0,C 180,E1 -23080.861,E2 -23080.861} C_VEL
LIN {X 0,Y 208.962,Z 413.418,A -85,B 0,C 180,E1 -23082.987,E2 -23082.987} C_VEL
LIN {X 0,Y 202.282,Z 423.821,A -85,B 0,C 180,E1 -23085.288,E2 -23085.288} C_VEL
LIN {X 0,Y 195.035,Z 434.043,A -85,B 0,C 180,E1 -23088.193,E2 -23088.193} C_VEL
LIN {X 0,Y 188.269,Z 442.609,A -85,B 0,C 180,E1 -23091.299,E2 -23091.299} C_VEL
LIN {X 0,Y 183.446,Z 448.413,A -85,B 0,C 180,E1 -23093.951,E2 -23093.951} C_VEL
LIN {X 0,Y 177.687,Z 454.918,A -85,B 0,C 180,E1 -23097.727,E2 -23097.727} C_VEL
LIN {X 0,Y 172.404,Z 460.542,A -85,B 0,C 180,E1 -23102.045,E2 -23102.045} C_VEL
LIN {X 0,Y 169.121,Z 463.936,A -85,B 0,C 180,E1 -23105.446,E2 -23105.446} C_VEL
LIN {X 0,Y 165.671,Z 467.335,A -85,B 0,C 180,E1 -23110.162,E2 -23110.162} C_VEL
LIN {X 0,Y 163.343,Z 469.591,A -85,B 0,C 180,E1 -23115.04,E2 -23115.04} C_VEL
LIN {X 0,Y 162.123,Z 470.752,A -85,B 0,C 180,E1 -23120.015,E2 -23120.015} C_VEL
LIN {X 0,Y 161.706,Z 470.807,A -85,B 0,C 180,E1 -23125.014,E2 -23125.014} C_VEL
LIN {X 0,Y 161.933,Z 469.679,A -85,B 0,C 180,E1 -23130.001,E2 -23130.001} C_VEL
LIN {X 0,Y 161.84,Z 467.347,A -85,B 0,C 180,E1 -23134.984,E2 -23134.984} C_VEL
LIN {X 0,Y 162.124,Z 463.754,A -85,B 0,C 180,E1 -23139.986,E2 -23139.986} C_VEL
LIN {X 0,Y 163.158,Z 458.802,A -85,B 0,C 180,E1 -23144.979,E2 -23144.979} C_VEL
LIN {X 0,Y 165.147,Z 452.358,A -85,B 0,C 180,E1 -23149.905,E2 -23149.905} C_VEL
LIN {X 0,Y 168.188,Z 444.24,A -85,B 0,C 180,E1 -23154.701,E2 -23154.701} C_VEL
LIN {X 0,Y 171.732,Z 435.561,A -85,B 0,C 180,E1 -23158.743,E2 -23158.743} C_VEL
LIN {X 0,Y 175.711,Z 425.619,A -85,B 0,C 180,E1 -23162.451,E2 -23162.451} C_VEL
LIN {X 0,Y 179.437,Z 416.249,A -85,B 0,C 180,E1 -23165.291,E2 -23165.291} C_VEL
LIN {X 0,Y 183.676,Z 404.822,A -85,B 0,C 180,E1 -23168.098,E2 -23168.098} C_VEL
LIN {X 0,Y 187.097,Z 395.071,A -85,B 0,C 180,E1 -23170.038,E2 -23170.038} C_VEL
LIN {X 0,Y 191.171,Z 382.156,A -85,B 0,C 180,E1 -23172.14,E2 -23172.14} C_VEL
LIN {X 0,Y 194.875,Z 368.437,A -85,B 0,C 180,E1 -23173.895,E2 -23173.895} C_VEL
LIN {X 0,Y 197.945,Z 354.776,A -85,B 0,C 180,E1 -23175.244,E2 -23175.244} C_VEL
LIN {X 0,Y 200.661,Z 339.472,A -85,B 0,C 180,E1 -23176.343,E2 -23176.343} C_VEL
LIN {X 0,Y 202.447,Z 325.094,A -85,B 0,C 180,E1 -23177.061,E2 -23177.061} C_VEL
LIN {X 0,Y 208.029,Z 241.97,A -85,B 0,C 180,E1 -23179.667,E2 -23179.667} C_VEL
LIN {X 0,Y 202.413,Z 227.117,A -85,B 0,C 180,E1 -23181.875,E2 -23181.875} C_VEL
LIN {X 0,Y 196.153,Z 212.879,A -85,B 0,C 180,E1 -23184.473,E2 -23184.473} C_VEL
LIN {X 0,Y 190.656,Z 201.956,A -85,B 0,C 180,E1 -23186.906,E2 -23186.906} C_VEL
LIN {X 0,Y 184.8,Z 193.176,A -85,B 0,C 180,E1 -23189.585,E2 -23189.585} C_VEL
LIN {X 0,Y 179.609,Z 185.751,A -85,B 0,C 180,E1 -23192.233,E2 -23192.233} C_VEL
LIN {X 0,Y 176.75,Z 181.824,A -85,B 0,C 180,E1 -23193.826,E2 -23193.826} C_VEL
LIN {X 0,Y 173.563,Z 177.941,A -85,B 0,C 180,E1 -23195.703,E2 -23195.703} C_VEL
LIN {X 0,Y 172.438,Z 176.28,A -85,B 0,C 180,E1 -23196.427,E2 -23196.427} C_VEL
LIN {X 0,Y 170.09,Z 173.878,A -85,B 0,C 180,E1 -23197.93,E2 -23197.93} C_VEL
LIN {X 0,Y 168.741,Z 171.301,A -85,B 0,C 180,E1 -23198.948,E2 -23198.948} C_VEL
LIN {X 0,Y 166.341,Z 169.561,A -85,B 0,C 180,E1 -23200.592,E2 -23200.592} C_VEL
LIN {X 0,Y 164.831,Z 167.083,A -85,B 0,C 180,E1 -23201.834,E2 -23201.834} C_VEL
LIN {X 0,Y 164.478,Z 165.609,A -85,B 0,C 180,E1 -23202.276,E2 -23202.276} C_VEL
LIN {X 0,Y 164.705,Z 165.587,A -85,B 0,C 180,E1 -23208.942,E2 -23208.942} C_VEL
LIN {X 0,Y 164.824,Z 165.567,A -85,B 0,C 180,E1 -23212.652,E2 -23212.652} C_VEL
LIN {X 0,Y 165.277,Z 165.469,A -85,B 0,C 180,E1 -23220.001,E2 -23220.001} C_VEL
LIN {X 0,Y 164.822,Z 165.537,A -85,B 0,C 180,E1 -23227.35,E2 -23227.35} C_VEL
LIN {X 0,Y 164.705,Z 165.545,A -85,B 0,C 180,E1 -23231.058,E2 -23231.058} C_VEL
LIN {X 0,Y 164.429,Z 165.614,A -85,B 0,C 180,E1 -23237.41,E2 -23237.41} C_VEL
LIN {X 0,Y 164.424,Z 165.628,A -85,B 0,C 180,E1 -23239.997,E2 -23239.997} C_VEL
LIN {X 0,Y 164.368,Z 165.619,A -85,B 0,C 180,E1 -23246.112,E2 -23246.112} C_VEL
LIN {X 0,Y 164.357,Z 165.596,A -85,B 0,C 180,E1 -23251.215,E2 -23251.215} C_VEL
LIN {X 0,Y 164.284,Z 165.609,A -85,B 0,C 180,E1 -23256.794,E2 -23256.794} C_VEL
LIN {X 0,Y 164.297,Z 165.633,A -85,B 0,C 180,E1 -23257.126,E2 -23257.126} C_VEL
LIN {X 0,Y 165.102,Z 168.074,A -85,B 0,C 180,E1 -23257.922,E2 -23257.922} C_VEL
LIN {X 0,Y 167.161,Z 170.488,A -85,B 0,C 180,E1 -23259.489,E2 -23259.489} C_VEL
LIN {X 0,Y 168.791,Z 171.577,A -85,B 0,C 180,E1 -23260.587,E2 -23260.587} C_VEL
LIN {X 0,Y 170.471,Z 174.561,A -85,B 0,C 180,E1 -23261.82,E2 -23261.82} C_VEL
LIN {X 0,Y 173.06,Z 177.141,A -85,B 0,C 180,E1 -23263.442,E2 -23263.442} C_VEL
LIN {X 0,Y 175.624,Z 180.678,A -85,B 0,C 180,E1 -23265.024,E2 -23265.024} C_VEL
LIN {X 0,Y 176.794,Z 182.02,A -85,B 0,C 180,E1 -23265.689,E2 -23265.689} C_VEL
LIN {X 0,Y 179.659,Z 185.857,A -85,B 0,C 180,E1 -23267.277,E2 -23267.277} C_VEL
LIN {X 0,Y 186.457,Z 195.541,A -85,B 0,C 180,E1 -23270.681,E2 -23270.681} C_VEL
LIN {X 0,Y 192.826,Z 205.413,A -85,B 0,C 180,E1 -23273.504,E2 -23273.504} C_VEL
LIN {X 0,Y 199.355,Z 216.855,A -85,B 0,C 180,E1 -23276.192,E2 -23276.192} C_VEL
LIN {X 0,Y 206.991,Z 231.806,A -85,B 0,C 180,E1 -23279.058,E2 -23279.058} C_VEL
LIN {X 0,Y 208.364,Z 235.183,A -85,B 0,C 180,E1 -23279.57,E2 -23279.57} C_VEL
LIN {X 0,Y 202.702,Z 316.754,A -85,B 0,C 180,E1 -23282.09,E2 -23282.09} C_VEL
LIN {X 0,Y 200.757,Z 332.693,A -85,B 0,C 180,E1 -23282.928,E2 -23282.928} C_VEL
LIN {X 0,Y 198.126,Z 347.869,A -85,B 0,C 180,E1 -23284.102,E2 -23284.102} C_VEL
LIN {X 0,Y 195.114,Z 361.558,A -85,B 0,C 180,E1 -23285.528,E2 -23285.528} C_VEL
LIN {X 0,Y 191.555,Z 375.024,A -85,B 0,C 180,E1 -23287.341,E2 -23287.341} C_VEL
LIN {X 0,Y 187.487,Z 388.176,A -85,B 0,C 180,E1 -23289.578,E2 -23289.578} C_VEL
LIN {X 0,Y 182.872,Z 401.237,A -85,B 0,C 180,E1 -23292.382,E2 -23292.382} C_VEL
LIN {X 0,Y 178.233,Z 413.405,A -85,B 0,C 180,E1 -23295.732,E2 -23295.732} C_VEL
LIN {X 0,Y 174.391,Z 422.843,A -85,B 0,C 180,E1 -23298.963,E2 -23298.963} C_VEL
LIN {X 0,Y 170.651,Z 432.074,A -85,B 0,C 180,E1 -23302.902,E2 -23302.902} C_VEL
LIN {X 0,Y 167.499,Z 439.759,A -85,B 0,C 180,E1 -23306.993,E2 -23306.993} C_VEL
LIN {X 0,Y 165.073,Z 446.118,A -85,B 0,C 180,E1 -23311.219,E2 -23311.219} C_VEL
LIN {X 0,Y 163.245,Z 451.777,A -85,B 0,C 180,E1 -23316.009,E2 -23316.009} C_VEL
LIN {X 0,Y 162.164,Z 455.454,A -85,B 0,C 180,E1 -23319.982,E2 -23319.982} C_VEL
LIN {X 0,Y 161.481,Z 458.908,A -85,B 0,C 180,E1 -23325.136,E2 -23325.136} C_VEL
LIN {X 0,Y 161.349,Z 461.114,A -85,B 0,C 180,E1 -23330.392,E2 -23330.392} C_VEL
LIN {X 0,Y 161.697,Z 461.944,A -85,B 0,C 180,E1 -23334.11,E2 -23334.11} C_VEL
LIN {X 0,Y 163.077,Z 461.862,A -85,B 0,C 180,E1 -23340.464,E2 -23340.464} C_VEL
LIN {X 0,Y 165.728,Z 460.153,A -85,B 0,C 180,E1 -23346.317,E2 -23346.317} C_VEL
LIN {X 0,Y 169.501,Z 456.996,A -85,B 0,C 180,E1 -23351.725,E2 -23351.725} C_VEL
LIN {X 0,Y 174.38,Z 452.409,A -85,B 0,C 180,E1 -23356.751,E2 -23356.751} C_VEL
LIN {X 0,Y 180.196,Z 446.514,A -85,B 0,C 180,E1 -23361.263,E2 -23361.263} C_VEL
LIN {X 0,Y 186.308,Z 439.711,A -85,B 0,C 180,E1 -23365.13,E2 -23365.13} C_VEL
LIN {X 0,Y 193.258,Z 431.338,A -85,B 0,C 180,E1 -23368.714,E2 -23368.714} C_VEL
LIN {X 0,Y 199.783,Z 422.702,A -85,B 0,C 180,E1 -23371.575,E2 -23371.575} C_VEL
LIN {X 0,Y 207.17,Z 411.756,A -85,B 0,C 180,E1 -23374.414,E2 -23374.414} C_VEL
LIN {X 0,Y 213.706,Z 400.854,A -85,B 0,C 180,E1 -23376.615,E2 -23376.615} C_VEL
LIN {X 0,Y 219.964,Z 388.928,A -85,B 0,C 180,E1 -23378.521,E2 -23378.521} C_VEL
LIN {X 0,Y 225.936,Z 375.548,A -85,B 0,C 180,E1 -23380.209,E2 -23380.209} C_VEL
LIN {X 0,Y 231.014,Z 361.911,A -85,B 0,C 180,E1 -23381.546,E2 -23381.546} C_VEL
LIN {X 0,Y 235.218,Z 347.872,A -85,B 0,C 180,E1 -23382.614,E2 -23382.614} C_VEL
LIN {X 0,Y 238.773,Z 332.734,A -85,B 0,C 180,E1 -23383.422,E2 -23383.422} C_VEL
LIN {X 0,Y 241.263,Z 317.202,A -85,B 0,C 180,E1 -23384.005,E2 -23384.005} C_VEL
LIN {X 0,Y 246.313,Z 261.818,A -85,B 0,C 180,E1 -23385.416,E2 -23385.416} C_VEL
LIN {X 0,Y 242.084,Z 253.839,A -85,B 0,C 180,E1 -23388.2,E2 -23388.2} C_VEL
LIN {X 0,Y 238.506,Z 247.526,A -85,B 0,C 180,E1 -23390.923,E2 -23390.923} C_VEL
LIN {X 0,Y 236.167,Z 243.595,A -85,B 0,C 180,E1 -23393.003,E2 -23393.003} C_VEL
LIN {X 0,Y 233.791,Z 239.578,A -85,B 0,C 180,E1 -23395.454,E2 -23395.454} C_VEL
LIN {X 0,Y 232.153,Z 236.785,A -85,B 0,C 180,E1 -23397.444,E2 -23397.444} C_VEL
LIN {X 0,Y 230.063,Z 233.84,A -85,B 0,C 180,E1 -23400.573,E2 -23400.573} C_VEL
LIN {X 0,Y 229.416,Z 232.115,A -85,B 0,C 180,E1 -23402.047,E2 -23402.047} C_VEL
LIN {X 0,Y 227.616,Z 230.465,A -85,B 0,C 180,E1 -23408.88,E2 -23408.88} C_VEL
LIN {X 0,Y 228.905,Z 232.117,A -85,B 0,C 180,E1 -23415.594,E2 -23415.594} C_VEL
LIN {X 0,Y 229.473,Z 232.777,A -85,B 0,C 180,E1 -23416.877,E2 -23416.877} C_VEL
LIN {X 0,Y 231.394,Z 236.273,A -85,B 0,C 180,E1 -23420.286,E2 -23420.286} C_VEL
LIN {X 0,Y 232.572,Z 238.121,A -85,B 0,C 180,E1 -23421.835,E2 -23421.835} C_VEL
LIN {X 0,Y 235.187,Z 243.377,A -85,B 0,C 180,E1 -23424.851,E2 -23424.851} C_VEL
LIN {X 0,Y 237.277,Z 247.558,A -85,B 0,C 180,E1 -23426.882,E2 -23426.882} C_VEL
LIN {X 0,Y 240.799,Z 254.958,A -85,B 0,C 180,E1 -23429.809,E2 -23429.809} C_VEL
LIN {X 0,Y 244.866,Z 264.66,A -85,B 0,C 180,E1 -23432.725,E2 -23432.725} C_VEL
LIN {X 0,Y 245.871,Z 267.189,A -85,B 0,C 180,E1 -23433.393,E2 -23433.393} C_VEL
LIN {X 0,Y 240.566,Z 325.149,A -85,B 0,C 180,E1 -23434.899,E2 -23434.899} C_VEL
LIN {X 0,Y 237.868,Z 340.733,A -85,B 0,C 180,E1 -23435.477,E2 -23435.477} C_VEL
LIN {X 0,Y 235.861,Z 349.193,A -85,B 0,C 180,E1 -23435.877,E2 -23435.877} C_VEL
LIN {X 0,Y 234.005,Z 354.791,A -85,B 0,C 180,E1 -23436.019,E2 -23436.019} C_VEL
LIN {X 0,Y 226.272,Z 370.86,A -85,B 0,C 180,E1 -23436.021,E2 -23436.021} C_VEL
LIN {X 0,Y 223.744,Z 376.107,A -85,B 0,C 180,E1 -23436.255,E2 -23436.255} C_VEL
LIN {X 0,Y 222.99,Z 377.819,A -85,B 0,C 180,E1 -23436.401,E2 -23436.401} C_VEL
LIN {X 0,Y 217.01,Z 391.234,A -85,B 0,C 180,E1 -23437.871,E2 -23437.871} C_VEL
LIN {X 0,Y 211.121,Z 402.549,A -85,B 0,C 180,E1 -23439.435,E2 -23439.435} C_VEL
LIN {X 0,Y 204.229,Z 414.281,A -85,B 0,C 180,E1 -23441.543,E2 -23441.543} C_VEL
LIN {X 0,Y 196.212,Z 426.101,A -85,B 0,C 180,E1 -23444.245,E2 -23444.245} C_VEL
LIN {X 0,Y 188.763,Z 435.903,A -85,B 0,C 180,E1 -23447.198,E2 -23447.198} C_VEL
LIN {X 0,Y 181.838,Z 444.089,A -85,B 0,C 180,E1 -23450.379,E2 -23450.379} C_VEL
LIN {X 0,Y 176.548,Z 450.03,A -85,B 0,C 180,E1 -23453.337,E2 -23453.337} C_VEL
LIN {X 0,Y 170.177,Z 456.634,A -85,B 0,C 180,E1 -23457.53,E2 -23457.53} C_VEL
LIN {X 0,Y 164.881,Z 461.859,A -85,B 0,C 180,E1 -23462.04,E2 -23462.04} C_VEL
LIN {X 0,Y 160.568,Z 465.807,A -85,B 0,C 180,E1 -23466.802,E2 -23466.802} C_VEL
LIN {X 0,Y 157.602,Z 468.543,A -85,B 0,C 180,E1 -23471.812,E2 -23471.812} C_VEL
LIN {X 0,Y 155.651,Z 470.166,A -85,B 0,C 180,E1 -23476.953,E2 -23476.953} C_VEL
LIN {X 0,Y 154.752,Z 470.704,A -85,B 0,C 180,E1 -23482.17,E2 -23482.17} C_VEL
LIN {X 0,Y 154.662,Z 470.124,A -85,B 0,C 180,E1 -23487.397,E2 -23487.397} C_VEL
LIN {X 0,Y 154.85,Z 469.379,A -85,B 0,C 180,E1 -23490.001,E2 -23490.001} C_VEL
LIN {X 0,Y 154.734,Z 466.963,A -85,B 0,C 180,E1 -23495.213,E2 -23495.213} C_VEL
LIN {X 0,Y 155.1,Z 463.284,A -85,B 0,C 180,E1 -23500.444,E2 -23500.444} C_VEL
LIN {X 0,Y 156.25,Z 458.238,A -85,B 0,C 180,E1 -23505.658,E2 -23505.658} C_VEL
LIN {X 0,Y 158.384,Z 451.691,A -85,B 0,C 180,E1 -23510.794,E2 -23510.794} C_VEL
LIN {X 0,Y 161.645,Z 443.463,A -85,B 0,C 180,E1 -23515.773,E2 -23515.773} C_VEL
LIN {X 0,Y 165.466,Z 434.667,A -85,B 0,C 180,E1 -23519.94,E2 -23519.94} C_VEL
LIN {X 0,Y 169.439,Z 425.042,A -85,B 0,C 180,E1 -23523.61,E2 -23523.61} C_VEL
LIN {X 0,Y 173.585,Z 415.059,A -85,B 0,C 180,E1 -23526.67,E2 -23526.67} C_VEL
LIN {X 0,Y 178.043,Z 403.48,A -85,B 0,C 180,E1 -23529.534,E2 -23529.534} C_VEL
LIN {X 0,Y 182.541,Z 390.884,A -85,B 0,C 180,E1 -23531.988,E2 -23531.988} C_VEL
LIN {X 0,Y 186.725,Z 377.653,A -85,B 0,C 180,E1 -23534.008,E2 -23534.008} C_VEL
LIN {X 0,Y 190.551,Z 362.69,A -85,B 0,C 180,E1 -23535.801,E2 -23535.801} C_VEL
LIN {X 0,Y 193.771,Z 347.95,A -85,B 0,C 180,E1 -23537.072,E2 -23537.072} C_VEL
LIN {X 0,Y 196.121,Z 332.688,A -85,B 0,C 180,E1 -23538.039,E2 -23538.039} C_VEL
LIN {X 0,Y 197.67,Z 317.125,A -85,B 0,C 180,E1 -23538.67,E2 -23538.67} C_VEL
LIN {X 0,Y 202.671,Z 243.85,A -85,B 0,C 180,E1 -23540.968,E2 -23540.968} C_VEL
LIN {X 0,Y 197.518,Z 230.127,A -85,B 0,C 180,E1 -23543.129,E2 -23543.129} C_VEL
LIN {X 0,Y 191.508,Z 216.184,A -85,B 0,C 180,E1 -23545.801,E2 -23545.801} C_VEL
LIN {X 0,Y 186.566,Z 206.338,A -85,B 0,C 180,E1 -23548.096,E2 -23548.096} C_VEL
LIN {X 0,Y 179.189,Z 195.164,A -85,B 0,C 180,E1 -23551.765,E2 -23551.765} C_VEL
LIN {X 0,Y 175.969,Z 190.739,A -85,B 0,C 180,E1 -23553.541,E2 -23553.541} C_VEL
LIN {X 0,Y 173.256,Z 186.966,A -85,B 0,C 180,E1 -23555.161,E2 -23555.161} C_VEL
LIN {X 0,Y 170.462,Z 183.161,A -85,B 0,C 180,E1 -23556.947,E2 -23556.947} C_VEL
LIN {X 0,Y 167.227,Z 179.349,A -85,B 0,C 180,E1 -23559.152,E2 -23559.152} C_VEL
LIN {X 0,Y 166.044,Z 177.526,A -85,B 0,C 180,E1 -23560.048,E2 -23560.048} C_VEL
LIN {X 0,Y 163.549,Z 175.058,A -85,B 0,C 180,E1 -23561.936,E2 -23561.936} C_VEL
LIN {X 0,Y 162.043,Z 172.289,A -85,B 0,C 180,E1 -23563.303,E2 -23563.303} C_VEL
LIN {X 0,Y 159.548,Z 170.706,A -85,B 0,C 180,E1 -23565.442,E2 -23565.442} C_VEL
LIN {X 0,Y 158.005,Z 168.369,A -85,B 0,C 180,E1 -23567.069,E2 -23567.069} C_VEL
LIN {X 0,Y 157.58,Z 166.47,A -85,B 0,C 180,E1 -23567.786,E2 -23567.786} C_VEL
LIN {X 0,Y 157.762,Z 166.447,A -85,B 0,C 180,E1 -23572.321,E2 -23572.321} C_VEL
LIN {X 0,Y 158.239,Z 166.345,A -85,B 0,C 180,E1 -23580.001,E2 -23580.001} C_VEL
LIN {X 0,Y 157.761,Z 166.412,A -85,B 0,C 180,E1 -23587.681,E2 -23587.681} C_VEL
LIN {X 0,Y 157.634,Z 166.426,A -85,B 0,C 180,E1 -23591.224,E2 -23591.224} C_VEL
LIN {X 0,Y 157.409,Z 166.495,A -85,B 0,C 180,E1 -23595.54,E2 -23595.54} C_VEL
LIN {X 0,Y 157.311,Z 166.505,A -85,B 0,C 180,E1 -23600.942,E2 -23600.942} C_VEL
LIN {X 0,Y 157.296,Z 166.487,A -85,B 0,C 180,E1 -23606.668,E2 -23606.668} C_VEL
LIN {X 0,Y 157.325,Z 166.645,A -85,B 0,C 180,E1 -23611.552,E2 -23611.552} C_VEL
LIN {X 0,Y 157.99,Z 168.822,A -85,B 0,C 180,E1 -23612.453,E2 -23612.453} C_VEL
LIN {X 0,Y 159.804,Z 171.122,A -85,B 0,C 180,E1 -23614.298,E2 -23614.298} C_VEL
LIN {X 0,Y 162.025,Z 172.5,A -85,B 0,C 180,E1 -23616.186,E2 -23616.186} C_VEL
LIN {X 0,Y 163.766,Z 175.612,A -85,B 0,C 180,E1 -23617.748,E2 -23617.748} C_VEL
LIN {X 0,Y 166.408,Z 178.019,A -85,B 0,C 180,E1 -23619.703,E2 -23619.703} C_VEL
LIN {X 0,Y 168.661,Z 181.445,A -85,B 0,C 180,E1 -23621.361,E2 -23621.361} C_VEL
LIN {X 0,Y 170.617,Z 183.508,A -85,B 0,C 180,E1 -23622.637,E2 -23622.637} C_VEL
LIN {X 0,Y 173.485,Z 187.242,A -85,B 0,C 180,E1 -23624.456,E2 -23624.456} C_VEL
LIN {X 0,Y 180.298,Z 196.854,A -85,B 0,C 180,E1 -23628.308,E2 -23628.308} C_VEL
LIN {X 0,Y 186.469,Z 206.203,A -85,B 0,C 180,E1 -23631.339,E2 -23631.339} C_VEL
LIN {X 0,Y 193.611,Z 218.381,A -85,B 0,C 180,E1 -23634.492,E2 -23634.492} C_VEL
LIN {X 0,Y 201.53,Z 233.891,A -85,B 0,C 180,E1 -23637.694,E2 -23637.694} C_VEL
LIN {X 0,Y 203.034,Z 237.42,A -85,B 0,C 180,E1 -23638.284,E2 -23638.284} C_VEL
LIN {X 0,Y 197.228,Z 317.728,A -85,B 0,C 180,E1 -23640.807,E2 -23640.807} C_VEL
LIN {X 0,Y 195.216,Z 333.382,A -85,B 0,C 180,E1 -23641.655,E2 -23641.655} C_VEL
LIN {X 0,Y 192.512,Z 348.419,A -85,B 0,C 180,E1 -23642.848,E2 -23642.848} C_VEL
LIN {X 0,Y 189.13,Z 362.963,A -85,B 0,C 180,E1 -23644.406,E2 -23644.406} C_VEL
LIN {X 0,Y 185.453,Z 376.243,A -85,B 0,C 180,E1 -23646.255,E2 -23646.255} C_VEL
LIN {X 0,Y 181.218,Z 389.297,A -85,B 0,C 180,E1 -23648.558,E2 -23648.558} C_VEL
LIN {X 0,Y 176.492,Z 402.099,A -85,B 0,C 180,E1 -23651.423,E2 -23651.423} C_VEL
LIN {X 0,Y 172.014,Z 413.324,A -85,B 0,C 180,E1 -23654.598,E2 -23654.598} C_VEL
LIN {X 0,Y 167.993,Z 422.786,A -85,B 0,C 180,E1 -23657.925,E2 -23657.925} C_VEL
LIN {X 0,Y 164.071,Z 432.058,A -85,B 0,C 180,E1 -23661.997,E2 -23661.997} C_VEL
LIN {X 0,Y 160.721,Z 439.785,A -85,B 0,C 180,E1 -23666.238,E2 -23666.238} C_VEL
LIN {X 0,Y 157.88,Z 447,A -85,B 0,C 180,E1 -23671.274,E2 -23671.274} C_VEL
LIN {X 0,Y 156.378,Z 451.404,A -85,B 0,C 180,E1 -23675.156,E2 -23675.156} C_VEL
LIN {X 0,Y 154.946,Z 456.066,A -85,B 0,C 180,E1 -23680.452,E2 -23680.452} C_VEL
LIN {X 0,Y 154.348,Z 459.415,A -85,B 0,C 180,E1 -23685.854,E2 -23685.854} C_VEL
LIN {X 0,Y 154.296,Z 461.502,A -85,B 0,C 180,E1 -23691.369,E2 -23691.369} C_VEL
LIN {X 0,Y 154.662,Z 462.147,A -85,B 0,C 180,E1 -23694.654,E2 -23694.654} C_VEL
LIN {X 0,Y 155.743,Z 462.25,A -85,B 0,C 180,E1 -23699.76,E2 -23699.76} C_VEL
LIN {X 0,Y 157.968,Z 461.133,A -85,B 0,C 180,E1 -23705.335,E2 -23705.335} C_VEL
LIN {X 0,Y 161.41,Z 458.664,A -85,B 0,C 180,E1 -23710.776,E2 -23710.776} C_VEL
LIN {X 0,Y 166.071,Z 454.762,A -85,B 0,C 180,E1 -23716.006,E2 -23716.006} C_VEL
LIN {X 0,Y 171.99,Z 449.326,A -85,B 0,C 180,E1 -23720.93,E2 -23720.93} C_VEL
LIN {X 0,Y 177.178,Z 444.132,A -85,B 0,C 180,E1 -23724.404,E2 -23724.404} C_VEL
LIN {X 0,Y 183.981,Z 436.743,A -85,B 0,C 180,E1 -23728.204,E2 -23728.204} C_VEL
LIN {X 0,Y 190.968,Z 428.503,A -85,B 0,C 180,E1 -23731.416,E2 -23731.416} C_VEL
LIN {X 0,Y 198.451,Z 418.553,A -85,B 0,C 180,E1 -23734.429,E2 -23734.429} C_VEL
LIN {X 0,Y 206.029,Z 407.16,A -85,B 0,C 180,E1 -23737.074,E2 -23737.074} C_VEL
LIN {X 0,Y 212.556,Z 396.064,A -85,B 0,C 180,E1 -23739.076,E2 -23739.076} C_VEL
LIN {X 0,Y 218.961,Z 383.377,A -85,B 0,C 180,E1 -23740.896,E2 -23740.896} C_VEL
LIN {X 0,Y 224.854,Z 369.583,A -85,B 0,C 180,E1 -23742.42,E2 -23742.42} C_VEL
LIN {X 0,Y 229.335,Z 356.807,A -85,B 0,C 180,E1 -23743.53,E2 -23743.53} C_VEL
LIN {X 0,Y 233.082,Z 343.559,A -85,B 0,C 180,E1 -23744.415,E2 -23744.415} C_VEL
LIN {X 0,Y 236.328,Z 328.719,A -85,B 0,C 180,E1 -23745.125,E2 -23745.125} C_VEL
LIN {X 0,Y 238.494,Z 313.598,A -85,B 0,C 180,E1 -23745.641,E2 -23745.641} C_VEL
LIN {X 0,Y 242.937,Z 265.597,A -85,B 0,C 180,E1 -23746.851,E2 -23746.851} C_VEL
LIN {X 0,Y 238.596,Z 257.266,A -85,B 0,C 180,E1 -23749.99,E2 -23749.99} C_VEL
LIN {X 0,Y 234.952,Z 250.672,A -85,B 0,C 180,E1 -23753.216,E2 -23753.216} C_VEL
LIN {X 0,Y 232.38,Z 246.199,A -85,B 0,C 180,E1 -23755.961,E2 -23755.961} C_VEL
LIN {X 0,Y 230.903,Z 243.581,A -85,B 0,C 180,E1 -23757.843,E2 -23757.843} C_VEL
LIN {X 0,Y 228.912,Z 240.615,A -85,B 0,C 180,E1 -23761.016,E2 -23761.016} C_VEL
LIN {X 0,Y 228.36,Z 239.097,A -85,B 0,C 180,E1 -23762.35,E2 -23762.35} C_VEL
LIN {X 0,Y 226.717,Z 237.512,A -85,B 0,C 180,E1 -23768.916,E2 -23768.916} C_VEL
LIN {X 0,Y 228.024,Z 239.211,A -85,B 0,C 180,E1 -23775.655,E2 -23775.655} C_VEL
LIN {X 0,Y 228.523,Z 240.005,A -85,B 0,C 180,E1 -23776.839,E2 -23776.839} C_VEL
LIN {X 0,Y 230.313,Z 243.212,A -85,B 0,C 180,E1 -23780.076,E2 -23780.076} C_VEL
LIN {X 0,Y 231.256,Z 244.913,A -85,B 0,C 180,E1 -23781.388,E2 -23781.388} C_VEL
LIN {X 0,Y 233.668,Z 249.952,A -85,B 0,C 180,E1 -23784.31,E2 -23784.31} C_VEL
LIN {X 0,Y 235.546,Z 253.948,A -85,B 0,C 180,E1 -23786.238,E2 -23786.238} C_VEL
LIN {X 0,Y 238.64,Z 260.82,A -85,B 0,C 180,E1 -23788.999,E2 -23788.999} C_VEL
LIN {X 0,Y 242.349,Z 270.049,A -85,B 0,C 180,E1 -23791.822,E2 -23791.822} C_VEL
LIN {X 0,Y 242.579,Z 270.673,A -85,B 0,C 180,E1 -23791.988,E2 -23791.988} C_VEL
LIN {X 0,Y 237.506,Z 324.275,A -85,B 0,C 180,E1 -23793.347,E2 -23793.347} C_VEL
LIN {X 0,Y 234.756,Z 340.078,A -85,B 0,C 180,E1 -23793.92,E2 -23793.92} C_VEL
LIN {X 0,Y 231.169,Z 354.404,A -85,B 0,C 180,E1 -23794.64,E2 -23794.64} C_VEL
LIN {X 0,Y 226.751,Z 368.005,A -85,B 0,C 180,E1 -23795.551,E2 -23795.551} C_VEL
LIN {X 0,Y 222.99,Z 377.819,A -85,B 0,C 180,E1 -23796.401,E2 -23796.401} C_VEL
LIN {X 0,Y 220.458,Z 383.035,A -85,B 0,C 180,E1 -23796.767,E2 -23796.767} C_VEL
LIN {X 0,Y 210.574,Z 397.72,A -85,B 0,C 180,E1 -23797.314,E2 -23797.314} C_VEL
LIN {X 0,Y 207.432,Z 402.411,A -85,B 0,C 180,E1 -23797.769,E2 -23797.769} C_VEL
LIN {X 0,Y 206.504,Z 403.928,A -85,B 0,C 180,E1 -23797.997,E2 -23797.997} C_VEL
LIN {X 0,Y 199.635,Z 415.105,A -85,B 0,C 180,E1 -23800.032,E2 -23800.032} C_VEL
LIN {X 0,Y 192.514,Z 425.197,A -85,B 0,C 180,E1 -23802.333,E2 -23802.333} C_VEL
LIN {X 0,Y 184.738,Z 435.107,A -85,B 0,C 180,E1 -23805.269,E2 -23805.269} C_VEL
LIN {X 0,Y 177.41,Z 443.396,A -85,B 0,C 180,E1 -23808.43,E2 -23808.43} C_VEL
LIN {X 0,Y 172.681,Z 448.397,A -85,B 0,C 180,E1 -23810.798,E2 -23810.798} C_VEL
LIN {X 0,Y 165.815,Z 455.343,A -85,B 0,C 180,E1 -23815.098,E2 -23815.098} C_VEL
LIN {X 0,Y 159.918,Z 460.765,A -85,B 0,C 180,E1 -23819.643,E2 -23819.643} C_VEL
LIN {X 0,Y 156.207,Z 464.022,A -85,B 0,C 180,E1 -23823.263,E2 -23823.263} C_VEL
LIN {X 0,Y 152.28,Z 467.299,A -85,B 0,C 180,E1 -23828.334,E2 -23828.334} C_VEL
LIN {X 0,Y 149.573,Z 469.39,A -85,B 0,C 180,E1 -23833.626,E2 -23833.626} C_VEL
LIN {X 0,Y 148.081,Z 470.39,A -85,B 0,C 180,E1 -23839.057,E2 -23839.057} C_VEL
LIN {X 0,Y 147.534,Z 470.301,A -85,B 0,C 180,E1 -23844.534,E2 -23844.534} C_VEL
LIN {X 0,Y 147.763,Z 469.078,A -85,B 0,C 180,E1 -23850.001,E2 -23850.001} C_VEL
LIN {X 0,Y 147.639,Z 466.58,A -85,B 0,C 180,E1 -23855.464,E2 -23855.464} C_VEL
LIN {X 0,Y 148.066,Z 462.812,A -85,B 0,C 180,E1 -23860.946,E2 -23860.946} C_VEL
LIN {X 0,Y 149.365,Z 457.675,A -85,B 0,C 180,E1 -23866.4,E2 -23866.4} C_VEL
LIN {X 0,Y 151.686,Z 451.027,A -85,B 0,C 180,E1 -23871.758,E2 -23871.758} C_VEL
LIN {X 0,Y 154.685,Z 443.831,A -85,B 0,C 180,E1 -23876.296,E2 -23876.296} C_VEL
LIN {X 0,Y 158.629,Z 435.154,A -85,B 0,C 180,E1 -23880.632,E2 -23880.632} C_VEL
LIN {X 0,Y 163.055,Z 424.951,A -85,B 0,C 180,E1 -23884.686,E2 -23884.686} C_VEL
LIN {X 0,Y 167.844,Z 413.853,A -85,B 0,C 180,E1 -23888.144,E2 -23888.144} C_VEL
LIN {X 0,Y 172.492,Z 402.061,A -85,B 0,C 180,E1 -23891.073,E2 -23891.073} C_VEL
LIN {X 0,Y 177.251,Z 389.225,A -85,B 0,C 180,E1 -23893.546,E2 -23893.546} C_VEL
LIN {X 0,Y 181.314,Z 376.663,A -85,B 0,C 180,E1 -23895.463,E2 -23895.463} C_VEL
LIN {X 0,Y 185.06,Z 362.467,A -85,B 0,C 180,E1 -23897.176,E2 -23897.176} C_VEL
LIN {X 0,Y 188.385,Z 347.72,A -85,B 0,C 180,E1 -23898.459,E2 -23898.459} C_VEL
LIN {X 0,Y 190.821,Z 332.449,A -85,B 0,C 180,E1 -23899.433,E2 -23899.433} C_VEL
LIN {X 0,Y 192.433,Z 316.558,A -85,B 0,C 180,E1 -23900.083,E2 -23900.083} C_VEL
LIN {X 0,Y 197.487,Z 246.08,A -85,B 0,C 180,E1 -23902.302,E2 -23902.302} C_VEL
LIN {X 0,Y 193.202,Z 234.342,A -85,B 0,C 180,E1 -23904.227,E2 -23904.227} C_VEL
LIN {X 0,Y 187.493,Z 220.801,A -85,B 0,C 180,E1 -23906.898,E2 -23906.898} C_VEL
LIN {X 0,Y 183.037,Z 211.589,A -85,B 0,C 180,E1 -23909.1,E2 -23909.1} C_VEL
LIN {X 0,Y 176.194,Z 200.917,A -85,B 0,C 180,E1 -23912.697,E2 -23912.697} C_VEL
LIN {X 0,Y 172.591,Z 195.87,A -85,B 0,C 180,E1 -23914.808,E2 -23914.808} C_VEL
LIN {X 0,Y 170.343,Z 192.662,A -85,B 0,C 180,E1 -23916.241,E2 -23916.241} C_VEL
LIN {X 0,Y 167.145,Z 188.352,A -85,B 0,C 180,E1 -23918.414,E2 -23918.414} C_VEL
LIN {X 0,Y 164.441,Z 184.816,A -85,B 0,C 180,E1 -23920.4,E2 -23920.4} C_VEL
LIN {X 0,Y 163.582,Z 183.742,A -85,B 0,C 180,E1 -23921.067,E2 -23921.067} C_VEL
LIN {X 0,Y 160.923,Z 180.592,A -85,B 0,C 180,E1 -23923.265,E2 -23923.265} C_VEL
LIN {X 0,Y 159.903,Z 178.872,A -85,B 0,C 180,E1 -23924.232,E2 -23924.232} C_VEL
LIN {X 0,Y 157.215,Z 176.614,A -85,B 0,C 180,E1 -23926.757,E2 -23926.757} C_VEL
LIN {X 0,Y 155.737,Z 173.785,A -85,B 0,C 180,E1 -23928.527,E2 -23928.527} C_VEL
LIN {X 0,Y 155.488,Z 173.207,A -85,B 0,C 180,E1 -23928.858,E2 -23928.858} C_VEL
LIN {X 0,Y 152.833,Z 171.58,A -85,B 0,C 180,E1 -23932.072,E2 -23932.072} C_VEL
LIN {X 0,Y 151.148,Z 169.234,A -85,B 0,C 180,E1 -23934.749,E2 -23934.749} C_VEL
LIN {X 0,Y 150.699,Z 167.322,A -85,B 0,C 180,E1 -23935.906,E2 -23935.906} C_VEL
LIN {X 0,Y 151.2,Z 167.221,A -85,B 0,C 180,E1 -23940.001,E2 -23940.001} C_VEL
LIN {X 0,Y 150.684,Z 167.288,A -85,B 0,C 180,E1 -23948.044,E2 -23948.044} C_VEL
LIN {X 0,Y 150.577,Z 167.306,A -85,B 0,C 180,E1 -23951.428,E2 -23951.428} C_VEL
LIN {X 0,Y 150.314,Z 167.373,A -85,B 0,C 180,E1 -23956.293,E2 -23956.293} C_VEL
LIN {X 0,Y 150.287,Z 167.382,A -85,B 0,C 180,E1 -23960.724,E2 -23960.724} C_VEL
LIN {X 0,Y 150.244,Z 167.562,A -85,B 0,C 180,E1 -23962.974,E2 -23962.974} C_VEL
LIN {X 0,Y 151.068,Z 169.944,A -85,B 0,C 180,E1 -23964.754,E2 -23964.754} C_VEL
LIN {X 0,Y 153.503,Z 172.524,A -85,B 0,C 180,E1 -23968.361,E2 -23968.361} C_VEL
LIN {X 0,Y 155.394,Z 173.389,A -85,B 0,C 180,E1 -23970.548,E2 -23970.548} C_VEL
LIN {X 0,Y 156.685,Z 176.183,A -85,B 0,C 180,E1 -23972.181,E2 -23972.181} C_VEL
LIN {X 0,Y 159.188,Z 178.55,A -85,B 0,C 180,E1 -23974.642,E2 -23974.642} C_VEL
LIN {X 0,Y 160.049,Z 179.273,A -85,B 0,C 180,E1 -23975.408,E2 -23975.408} C_VEL
LIN {X 0,Y 162.29,Z 182.696,A -85,B 0,C 180,E1 -23977.425,E2 -23977.425} C_VEL
LIN {X 0,Y 164.294,Z 184.716,A -85,B 0,C 180,E1 -23978.976,E2 -23978.976} C_VEL
LIN {X 0,Y 166.914,Z 188.316,A -85,B 0,C 180,E1 -23980.925,E2 -23980.925} C_VEL
LIN {X 0,Y 168.197,Z 189.783,A -85,B 0,C 180,E1 -23981.8,E2 -23981.8} C_VEL
LIN {X 0,Y 171.78,Z 194.777,A -85,B 0,C 180,E1 -23984.169,E2 -23984.169} C_VEL
LIN {X 0,Y 176.994,Z 202.152,A -85,B 0,C 180,E1 -23987.231,E2 -23987.231} C_VEL
LIN {X 0,Y 183.415,Z 212.25,A -85,B 0,C 180,E1 -23990.566,E2 -23990.566} C_VEL
LIN {X 0,Y 190.049,Z 223.913,A -85,B 0,C 180,E1 -23993.633,E2 -23993.633} C_VEL
LIN {X 0,Y 197.714,Z 239.359,A -85,B 0,C 180,E1 -23996.886,E2 -23996.886} C_VEL
LIN {X 0,Y 194.146,Z 289.435,A -85,B 0,C 180,E1 -23998.468,E2 -23998.468} C_VEL
LIN {X 0,Y 191.869,Z 318.644,A -85,B 0,C 180,E1 -23999.453,E2 -23999.453} C_VEL
LIN {X 0,Y 189.794,Z 334.056,A -85,B 0,C 180,E1 -24000.311,E2 -24000.311} C_VEL
LIN {X 0,Y 186.977,Z 348.98,A -85,B 0,C 180,E1 -24001.516,E2 -24001.516} C_VEL
LIN {X 0,Y 183.719,Z 362.561,A -85,B 0,C 180,E1 -24002.981,E2 -24002.981} C_VEL
LIN {X 0,Y 179.892,Z 375.933,A -85,B 0,C 180,E1 -24004.857,E2 -24004.857} C_VEL
LIN {X 0,Y 175.62,Z 388.724,A -85,B 0,C 180,E1 -24007.137,E2 -24007.137} C_VEL
LIN {X 0,Y 170.971,Z 400.901,A -85,B 0,C 180,E1 -24009.862,E2 -24009.862} C_VEL
LIN {X 0,Y 166.592,Z 411.449,A -85,B 0,C 180,E1 -24012.823,E2 -24012.823} C_VEL
LIN {X 0,Y 162.308,Z 421.227,A -85,B 0,C 180,E1 -24016.221,E2 -24016.221} C_VEL
LIN {X 0,Y 158.027,Z 430.805,A -85,B 0,C 180,E1 -24020.399,E2 -24020.399} C_VEL
LIN {X 0,Y 154.476,Z 438.779,A -85,B 0,C 180,E1 -24024.778,E2 -24024.778} C_VEL
LIN {X 0,Y 151.283,Z 446.236,A -85,B 0,C 180,E1 -24029.999,E2 -24029.999} C_VEL
LIN {X 0,Y 149.16,Z 452.134,A -85,B 0,C 180,E1 -24035.406,E2 -24035.406} C_VEL
LIN {X 0,Y 147.726,Z 456.655,A -85,B 0,C 180,E1 -24040.969,E2 -24040.969} C_VEL
LIN {X 0,Y 147.208,Z 459.868,A -85,B 0,C 180,E1 -24046.645,E2 -24046.645} C_VEL
LIN {X 0,Y 147.288,Z 461.842,A -85,B 0,C 180,E1 -24052.44,E2 -24052.44} C_VEL
LIN {X 0,Y 147.652,Z 462.358,A -85,B 0,C 180,E1 -24055.364,E2 -24055.364} C_VEL
LIN {X 0,Y 149.071,Z 462.424,A -85,B 0,C 180,E1 -24061.237,E2 -24061.237} C_VEL
LIN {X 0,Y 151.674,Z 461.165,A -85,B 0,C 180,E1 -24067.039,E2 -24067.039} C_VEL
LIN {X 0,Y 155.566,Z 458.545,A -85,B 0,C 180,E1 -24072.659,E2 -24072.659} C_VEL
LIN {X 0,Y 160.711,Z 454.486,A -85,B 0,C 180,E1 -24078.023,E2 -24078.023} C_VEL
LIN {X 0,Y 167.142,Z 448.901,A -85,B 0,C 180,E1 -24083.025,E2 -24083.025} C_VEL
LIN {X 0,Y 172.726,Z 443.553,A -85,B 0,C 180,E1 -24086.523,E2 -24086.523} C_VEL
LIN {X 0,Y 179.985,Z 435.988,A -85,B 0,C 180,E1 -24090.32,E2 -24090.32} C_VEL
LIN {X 0,Y 188.017,Z 426.735,A -85,B 0,C 180,E1 -24093.779,E2 -24093.779} C_VEL
LIN {X 0,Y 196.033,Z 416.233,A -85,B 0,C 180,E1 -24096.773,E2 -24096.773} C_VEL
LIN {X 0,Y 203.154,Z 405.701,A -85,B 0,C 180,E1 -24099.073,E2 -24099.073} C_VEL
LIN {X 0,Y 209.926,Z 394.265,A -85,B 0,C 180,E1 -24101.042,E2 -24101.042} C_VEL
LIN {X 0,Y 216.021,Z 382.314,A -85,B 0,C 180,E1 -24102.687,E2 -24102.687} C_VEL
LIN {X 0,Y 221.913,Z 368.66,A -85,B 0,C 180,E1 -24104.148,E2 -24104.148} C_VEL
LIN {X 0,Y 226.888,Z 354.562,A -85,B 0,C 180,E1 -24105.301,E2 -24105.301} C_VEL
LIN {X 0,Y 230.535,Z 341.67,A -85,B 0,C 180,E1 -24106.106,E2 -24106.106} C_VEL
LIN {X 0,Y 233.82,Z 326.173,A -85,B 0,C 180,E1 -24106.794,E2 -24106.794} C_VEL
LIN {X 0,Y 235.977,Z 309.655,A -85,B 0,C 180,E1 -24107.297,E2 -24107.297} C_VEL
LIN {X 0,Y 239.771,Z 269.592,A -85,B 0,C 180,E1 -24108.278,E2 -24108.278} C_VEL
LIN {X 0,Y 235.94,Z 262.037,A -85,B 0,C 180,E1 -24111.346,E2 -24111.346} C_VEL
LIN {X 0,Y 232.974,Z 256.521,A -85,B 0,C 180,E1 -24114.199,E2 -24114.199} C_VEL
LIN {X 0,Y 230.885,Z 252.67,A -85,B 0,C 180,E1 -24116.598,E2 -24116.598} C_VEL
LIN {X 0,Y 229.533,Z 250.306,A -85,B 0,C 180,E1 -24118.409,E2 -24118.409} C_VEL
LIN {X 0,Y 227.696,Z 247.153,A -85,B 0,C 180,E1 -24121.657,E2 -24121.657} C_VEL
LIN {X 0,Y 227.312,Z 246.07,A -85,B 0,C 180,E1 -24122.656,E2 -24122.656} C_VEL
LIN {X 0,Y 225.817,Z 244.563,A -85,B 0,C 180,E1 -24128.952,E2 -24128.952} C_VEL
LIN {X 0,Y 227.238,Z 246.379,A -85,B 0,C 180,E1 -24135.936,E2 -24135.936} C_VEL
LIN {X 0,Y 229.729,Z 251.117,A -85,B 0,C 180,E1 -24140.595,E2 -24140.595} C_VEL
LIN {X 0,Y 232.126,Z 256.434,A -85,B 0,C 180,E1 -24143.71,E2 -24143.71} C_VEL
LIN {X 0,Y 233.706,Z 259.96,A -85,B 0,C 180,E1 -24145.435,E2 -24145.435} C_VEL
LIN {X 0,Y 236.761,Z 267.227,A -85,B 0,C 180,E1 -24148.355,E2 -24148.355} C_VEL
LIN {X 0,Y 239.391,Z 274.111,A -85,B 0,C 180,E1 -24150.516,E2 -24150.516} C_VEL
LIN {X 0,Y 234.465,Z 324.465,A -85,B 0,C 180,E1 -24151.789,E2 -24151.789} C_VEL
LIN {X 0,Y 231.636,Z 340.172,A -85,B 0,C 180,E1 -24152.351,E2 -24152.351} C_VEL
LIN {X 0,Y 227.634,Z 355.55,A -85,B 0,C 180,E1 -24153.128,E2 -24153.128} C_VEL
LIN {X 0,Y 223.45,Z 367.996,A -85,B 0,C 180,E1 -24153.948,E2 -24153.948} C_VEL
LIN {X 0,Y 218.041,Z 381.352,A -85,B 0,C 180,E1 -24155.126,E2 -24155.126} C_VEL
LIN {X 0,Y 212.108,Z 393.707,A -85,B 0,C 180,E1 -24156.535,E2 -24156.535} C_VEL
LIN {X 0,Y 206.504,Z 403.928,A -85,B 0,C 180,E1 -24157.997,E2 -24157.997} C_VEL
LIN {X 0,Y 203.45,Z 408.523,A -85,B 0,C 180,E1 -24158.616,E2 -24158.616} C_VEL
LIN {X 0,Y 197.156,Z 415.809,A -85,B 0,C 180,E1 -24159.312,E2 -24159.312} C_VEL
LIN {X 0,Y 190.635,Z 422.734,A -85,B 0,C 180,E1 -24160.126,E2 -24160.126} C_VEL
LIN {X 0,Y 187.192,Z 426.654,A -85,B 0,C 180,E1 -24160.96,E2 -24160.96} C_VEL
LIN {X 0,Y 179.776,Z 435.638,A -85,B 0,C 180,E1 -24163.68,E2 -24163.68} C_VEL
LIN {X 0,Y 172.159,Z 443.81,A -85,B 0,C 180,E1 -24166.861,E2 -24166.861} C_VEL
LIN {X 0,Y 166.872,Z 449.051,A -85,B 0,C 180,E1 -24169.445,E2 -24169.445} C_VEL
LIN {X 0,Y 160.027,Z 455.571,A -85,B 0,C 180,E1 -24173.639,E2 -24173.639} C_VEL
LIN {X 0,Y 153.808,Z 460.904,A -85,B 0,C 180,E1 -24178.301,E2 -24178.301} C_VEL
LIN {X 0,Y 149.862,Z 464.057,A -85,B 0,C 180,E1 -24182.034,E2 -24182.034} C_VEL
LIN {X 0,Y 145.634,Z 467.266,A -85,B 0,C 180,E1 -24187.291,E2 -24187.291} C_VEL
LIN {X 0,Y 142.734,Z 469.29,A -85,B 0,C 180,E1 -24192.818,E2 -24192.818} C_VEL
LIN {X 0,Y 141.076,Z 470.209,A -85,B 0,C 180,E1 -24198.507,E2 -24198.507} C_VEL
LIN {X 0,Y 140.442,Z 470.039,A -85,B 0,C 180,E1 -24204.257,E2 -24204.257} C_VEL
LIN {X 0,Y 140.686,Z 468.755,A -85,B 0,C 180,E1 -24210.001,E2 -24210.001} C_VEL
LIN {X 0,Y 140.547,Z 466.196,A -85,B 0,C 180,E1 -24215.741,E2 -24215.741} C_VEL
LIN {X 0,Y 141.054,Z 462.342,A -85,B 0,C 180,E1 -24221.497,E2 -24221.497} C_VEL
LIN {X 0,Y 142.479,Z 457.109,A -85,B 0,C 180,E1 -24227.216,E2 -24227.216} C_VEL
LIN {X 0,Y 145.287,Z 449.823,A -85,B 0,C 180,E1 -24233.209,E2 -24233.209} C_VEL
LIN {X 0,Y 148.811,Z 441.918,A -85,B 0,C 180,E1 -24238.184,E2 -24238.184} C_VEL
LIN {X 0,Y 153.11,Z 432.871,A -85,B 0,C 180,E1 -24242.64,E2 -24242.64} C_VEL
LIN {X 0,Y 157.319,Z 423.505,A -85,B 0,C 180,E1 -24246.336,E2 -24246.336} C_VEL
LIN {X 0,Y 162.226,Z 412.649,A -85,B 0,C 180,E1 -24249.719,E2 -24249.719} C_VEL
LIN {X 0,Y 167.108,Z 400.651,A -85,B 0,C 180,E1 -24252.702,E2 -24252.702} C_VEL
LIN {X 0,Y 171.587,Z 389.012,A -85,B 0,C 180,E1 -24254.955,E2 -24254.955} C_VEL
LIN {X 0,Y 176.063,Z 375.543,A -85,B 0,C 180,E1 -24257.019,E2 -24257.019} C_VEL
LIN {X 0,Y 179.96,Z 361.102,A -85,B 0,C 180,E1 -24258.746,E2 -24258.746} C_VEL
LIN {X 0,Y 183.259,Z 346.723,A -85,B 0,C 180,E1 -24259.98,E2 -24259.98} C_VEL
LIN {X 0,Y 185.791,Z 331.075,A -85,B 0,C 180,E1 -24260.956,E2 -24260.956} C_VEL
LIN {X 0,Y 187.438,Z 314.508,A -85,B 0,C 180,E1 -24261.619,E2 -24261.619} C_VEL
LIN {X 0,Y 192.358,Z 248.146,A -85,B 0,C 180,E1 -24263.734,E2 -24263.734} C_VEL
LIN {X 0,Y 187.922,Z 235.783,A -85,B 0,C 180,E1 -24265.878,E2 -24265.878} C_VEL
LIN {X 0,Y 181.768,Z 221.366,A -85,B 0,C 180,E1 -24268.971,E2 -24268.971} C_VEL
LIN {X 0,Y 178.75,Z 215.51,A -85,B 0,C 180,E1 -24270.569,E2 -24270.569} C_VEL
LIN {X 0,Y 172.594,Z 205.727,A -85,B 0,C 180,E1 -24274.052,E2 -24274.052} C_VEL
LIN {X 0,Y 167.585,Z 198.483,A -85,B 0,C 180,E1 -24277.292,E2 -24277.292} C_VEL
LIN {X 0,Y 164.65,Z 194.455,A -85,B 0,C 180,E1 -24279.382,E2 -24279.382} C_VEL
LIN {X 0,Y 161.381,Z 190.023,A -85,B 0,C 180,E1 -24281.96,E2 -24281.96} C_VEL
LIN {X 0,Y 158.785,Z 186.769,A -85,B 0,C 180,E1 -24284.239,E2 -24284.239} C_VEL
LIN {X 0,Y 157.84,Z 185.354,A -85,B 0,C 180,E1 -24285.167,E2 -24285.167} C_VEL
LIN {X 0,Y 155.212,Z 182.815,A -85,B 0,C 180,E1 -24287.832,E2 -24287.832} C_VEL
LIN {X 0,Y 153.687,Z 179.927,A -85,B 0,C 180,E1 -24289.794,E2 -24289.794} C_VEL
LIN {X 0,Y 151.026,Z 177.903,A -85,B 0,C 180,E1 -24293.32,E2 -24293.32} C_VEL
LIN {X 0,Y 149.553,Z 175.38,A -85,B 0,C 180,E1 -24295.959,E2 -24295.959} C_VEL
LIN {X 0,Y 149.11,Z 174.185,A -85,B 0,C 180,E1 -24296.962,E2 -24296.962} C_VEL
LIN {X 0,Y 147.221,Z 173.27,A -85,B 0,C 180,E1 -24301.232,E2 -24301.232} C_VEL
LIN {X 0,Y 145.834,Z 172.497,A -85,B 0,C 180,E1 -24308.314,E2 -24308.314} C_VEL
LIN {X 0,Y 145.994,Z 172.901,A -85,B 0,C 180,E1 -24313.219,E2 -24313.219} C_VEL
LIN {X 0,Y 148.923,Z 174.576,A -85,B 0,C 180,E1 -24322.274,E2 -24322.274} C_VEL
LIN {X 0,Y 149.999,Z 177.156,A -85,B 0,C 180,E1 -24324.573,E2 -24324.573} C_VEL
LIN {X 0,Y 152.434,Z 179.545,A -85,B 0,C 180,E1 -24328.203,E2 -24328.203} C_VEL
LIN {X 0,Y 153.757,Z 180.349,A -85,B 0,C 180,E1 -24329.818,E2 -24329.818} C_VEL
LIN {X 0,Y 155.536,Z 183.495,A -85,B 0,C 180,E1 -24332.044,E2 -24332.044} C_VEL
LIN {X 0,Y 158.149,Z 185.935,A -85,B 0,C 180,E1 -24334.636,E2 -24334.636} C_VEL
LIN {X 0,Y 160.559,Z 189.433,A -85,B 0,C 180,E1 -24336.874,E2 -24336.874} C_VEL
LIN {X 0,Y 162.046,Z 191.067,A -85,B 0,C 180,E1 -24338.088,E2 -24338.088} C_VEL
LIN {X 0,Y 164.995,Z 194.974,A -85,B 0,C 180,E1 -24340.361,E2 -24340.361} C_VEL
LIN {X 0,Y 169.014,Z 200.598,A -85,B 0,C 180,E1 -24343.161,E2 -24343.161} C_VEL
LIN {X 0,Y 174.229,Z 208.248,A -85,B 0,C 180,E1 -24346.397,E2 -24346.397} C_VEL
LIN {X 0,Y 180.12,Z 217.823,A -85,B 0,C 180,E1 -24349.625,E2 -24349.625} C_VEL
LIN {X 0,Y 186.109,Z 228.66,A -85,B 0,C 180,E1 -24352.56,E2 -24352.56} C_VEL
LIN {X 0,Y 192.66,Z 241.984,A -85,B 0,C 180,E1 -24355.495,E2 -24355.495} C_VEL
LIN {X 0,Y 186.8,Z 318.013,A -85,B 0,C 180,E1 -24357.945,E2 -24357.945} C_VEL
LIN {X 0,Y 184.59,Z 333.996,A -85,B 0,C 180,E1 -24358.83,E2 -24358.83} C_VEL
LIN {X 0,Y 181.821,Z 348.411,A -85,B 0,C 180,E1 -24359.994,E2 -24359.994} C_VEL
LIN {X 0,Y 178.434,Z 362.124,A -85,B 0,C 180,E1 -24361.472,E2 -24361.472} C_VEL
LIN {X 0,Y 174.459,Z 375.592,A -85,B 0,C 180,E1 -24363.373,E2 -24363.373} C_VEL
LIN {X 0,Y 169.806,Z 389.04,A -85,B 0,C 180,E1 -24365.799,E2 -24365.799} C_VEL
LIN {X 0,Y 164.717,Z 401.808,A -85,B 0,C 180,E1 -24368.735,E2 -24368.735} C_VEL
LIN {X 0,Y 159.816,Z 413.133,A -85,B 0,C 180,E1 -24372.07,E2 -24372.07} C_VEL
LIN {X 0,Y 154.695,Z 424.151,A -85,B 0,C 180,E1 -24376.2,E2 -24376.2} C_VEL
LIN {X 0,Y 150.44,Z 433.271,A -85,B 0,C 180,E1 -24380.588,E2 -24380.588} C_VEL
LIN {X 0,Y 146.816,Z 440.862,A -85,B 0,C 180,E1 -24385.194,E2 -24385.194} C_VEL
LIN {X 0,Y 144.061,Z 447.122,A -85,B 0,C 180,E1 -24389.999,E2 -24389.999} C_VEL
LIN {X 0,Y 141.931,Z 452.867,A -85,B 0,C 180,E1 -24395.682,E2 -24395.682} C_VEL
LIN {X 0,Y 140.535,Z 457.244,A -85,B 0,C 180,E1 -24401.538,E2 -24401.538} C_VEL
LIN {X 0,Y 140.058,Z 460.337,A -85,B 0,C 180,E1 -24407.555,E2 -24407.555} C_VEL
LIN {X 0,Y 140.308,Z 462.159,A -85,B 0,C 180,E1 -24413.622,E2 -24413.622} C_VEL
LIN {X 0,Y 141.454,Z 462.735,A -85,B 0,C 180,E1 -24419.79,E2 -24419.79} C_VEL
LIN {X 0,Y 143.817,Z 462.013,A -85,B 0,C 180,E1 -24425.901,E2 -24425.901} C_VEL
LIN {X 0,Y 147.554,Z 459.956,A -85,B 0,C 180,E1 -24431.821,E2 -24431.821} C_VEL
LIN {X 0,Y 152.551,Z 456.494,A -85,B 0,C 180,E1 -24437.485,E2 -24437.485} C_VEL
LIN {X 0,Y 158.904,Z 451.528,A -85,B 0,C 180,E1 -24442.758,E2 -24442.758} C_VEL
LIN {X 0,Y 166.468,Z 444.915,A -85,B 0,C 180,E1 -24447.603,E2 -24447.603} C_VEL
LIN {X 0,Y 173.478,Z 438.16,A -85,B 0,C 180,E1 -24451.236,E2 -24451.236} C_VEL
LIN {X 0,Y 181.325,Z 429.757,A -85,B 0,C 180,E1 -24454.627,E2 -24454.627} C_VEL
LIN {X 0,Y 189.809,Z 419.475,A -85,B 0,C 180,E1 -24457.767,E2 -24457.767} C_VEL
LIN {X 0,Y 197.773,Z 408.427,A -85,B 0,C 180,E1 -24460.336,E2 -24460.336} C_VEL
LIN {X 0,Y 205.175,Z 396.698,A -85,B 0,C 180,E1 -24462.42,E2 -24462.42} C_VEL
LIN {X 0,Y 211.853,Z 384.304,A -85,B 0,C 180,E1 -24464.161,E2 -24464.161} C_VEL
LIN {X 0,Y 217.721,Z 371.475,A -85,B 0,C 180,E1 -24465.555,E2 -24465.555} C_VEL
LIN {X 0,Y 222.936,Z 357.603,A -85,B 0,C 180,E1 -24466.734,E2 -24466.734} C_VEL
LIN {X 0,Y 226.984,Z 344.112,A -85,B 0,C 180,E1 -24467.605,E2 -24467.605} C_VEL
LIN {X 0,Y 230.47,Z 328.891,A -85,B 0,C 180,E1 -24468.305,E2 -24468.305} C_VEL
LIN {X 0,Y 232.773,Z 313.482,A -85,B 0,C 180,E1 -24468.803,E2 -24468.803} C_VEL
LIN {X 0,Y 236.701,Z 273.579,A -85,B 0,C 180,E1 -24469.783,E2 -24469.783} C_VEL
LIN {X 0,Y 233.394,Z 266.759,A -85,B 0,C 180,E1 -24472.757,E2 -24472.757} C_VEL
LIN {X 0,Y 231.125,Z 262.494,A -85,B 0,C 180,E1 -24475.129,E2 -24475.129} C_VEL
LIN {X 0,Y 229.582,Z 259.464,A -85,B 0,C 180,E1 -24477.025,E2 -24477.025} C_VEL
LIN {X 0,Y 228.25,Z 257.075,A -85,B 0,C 180,E1 -24478.895,E2 -24478.895} C_VEL
LIN {X 0,Y 226.468,Z 253.534,A -85,B 0,C 180,E1 -24482.425,E2 -24482.425} C_VEL
LIN {X 0,Y 226.032,Z 252.824,A -85,B 0,C 180,E1 -24483.565,E2 -24483.565} C_VEL
LIN {X 0,Y 224.92,Z 251.593,A -85,B 0,C 180,E1 -24488.988,E2 -24488.988} C_VEL
LIN {X 0,Y 226.246,Z 253.382,A -85,B 0,C 180,E1 -24495.737,E2 -24495.737} C_VEL
LIN {X 0,Y 228.449,Z 257.898,A -85,B 0,C 180,E1 -24500.13,E2 -24500.13} C_VEL
LIN {X 0,Y 230.605,Z 262.936,A -85,B 0,C 180,E1 -24503.099,E2 -24503.099} C_VEL
LIN {X 0,Y 232.255,Z 266.835,A -85,B 0,C 180,E1 -24505.002,E2 -24505.002} C_VEL
LIN {X 0,Y 235.126,Z 274.182,A -85,B 0,C 180,E1 -24507.887,E2 -24507.887} C_VEL
LIN {X 0,Y 236.361,Z 277.655,A -85,B 0,C 180,E1 -24509.012,E2 -24509.012} C_VEL
LIN {X 0,Y 231.744,Z 323.806,A -85,B 0,C 180,E1 -24510.173,E2 -24510.173} C_VEL
LIN {X 0,Y 228.887,Z 339.513,A -85,B 0,C 180,E1 -24510.713,E2 -24510.713} C_VEL
LIN {X 0,Y 224.94,Z 354.472,A -85,B 0,C 180,E1 -24511.423,E2 -24511.423} C_VEL
LIN {X 0,Y 220.326,Z 367.988,A -85,B 0,C 180,E1 -24512.297,E2 -24512.297} C_VEL
LIN {X 0,Y 214.777,Z 381.308,A -85,B 0,C 180,E1 -24513.446,E2 -24513.446} C_VEL
LIN {X 0,Y 208.012,Z 394.905,A -85,B 0,C 180,E1 -24514.984,E2 -24514.984} C_VEL
LIN {X 0,Y 202.316,Z 404.791,A -85,B 0,C 180,E1 -24516.413,E2 -24516.413} C_VEL
LIN {X 0,Y 195.186,Z 415.875,A -85,B 0,C 180,E1 -24518.452,E2 -24518.452} C_VEL
LIN {X 0,Y 187.192,Z 426.654,A -85,B 0,C 180,E1 -24520.96,E2 -24520.96} C_VEL
LIN {X 0,Y 183.69,Z 430.516,A -85,B 0,C 180,E1 -24521.862,E2 -24521.862} C_VEL
LIN {X 0,Y 176.726,Z 436.486,A -85,B 0,C 180,E1 -24523.047,E2 -24523.047} C_VEL
LIN {X 0,Y 169.677,Z 442.04,A -85,B 0,C 180,E1 -24524.417,E2 -24524.417} C_VEL
LIN {X 0,Y 166.104,Z 445.103,A -85,B 0,C 180,E1 -24525.622,E2 -24525.622} C_VEL
LIN {X 0,Y 159.842,Z 450.919,A -85,B 0,C 180,E1 -24528.737,E2 -24528.737} C_VEL
LIN {X 0,Y 152.559,Z 457.185,A -85,B 0,C 180,E1 -24533.212,E2 -24533.212} C_VEL
LIN {X 0,Y 146.298,Z 462.106,A -85,B 0,C 180,E1 -24538.102,E2 -24538.102} C_VEL
LIN {X 0,Y 141.128,Z 465.805,A -85,B 0,C 180,E1 -24543.374,E2 -24543.374} C_VEL
LIN {X 0,Y 137.316,Z 468.357,A -85,B 0,C 180,E1 -24549.007,E2 -24549.007} C_VEL
LIN {X 0,Y 134.799,Z 469.744,A -85,B 0,C 180,E1 -24554.89,E2 -24554.89} C_VEL
LIN {X 0,Y 133.589,Z 470.041,A -85,B 0,C 180,E1 -24560.92,E2 -24560.92} C_VEL
LIN {X 0,Y 133.387,Z 469.239,A -85,B 0,C 180,E1 -24566.981,E2 -24566.981} C_VEL
LIN {X 0,Y 133.539,Z 468.164,A -85,B 0,C 180,E1 -24570.679,E2 -24570.679} C_VEL
LIN {X 0,Y 133.451,Z 465.805,A -85,B 0,C 180,E1 -24576.047,E2 -24576.047} C_VEL
LIN {X 0,Y 134.043,Z 461.87,A -85,B 0,C 180,E1 -24582.107,E2 -24582.107} C_VEL
LIN {X 0,Y 135.637,Z 456.545,A -85,B 0,C 180,E1 -24588.114,E2 -24588.114} C_VEL
LIN {X 0,Y 138.435,Z 449.699,A -85,B 0,C 180,E1 -24593.964,E2 -24593.964} C_VEL
LIN {X 0,Y 142.484,Z 441.142,A -85,B 0,C 180,E1 -24599.556,E2 -24599.556} C_VEL
LIN {X 0,Y 147.09,Z 431.975,A -85,B 0,C 180,E1 -24604.155,E2 -24604.155} C_VEL
LIN {X 0,Y 151.923,Z 421.881,A -85,B 0,C 180,E1 -24608.149,E2 -24608.149} C_VEL
LIN {X 0,Y 157.176,Z 410.444,A -85,B 0,C 180,E1 -24611.693,E2 -24611.693} C_VEL
LIN {X 0,Y 162.38,Z 398.048,A -85,B 0,C 180,E1 -24614.696,E2 -24614.696} C_VEL
LIN {X 0,Y 167.048,Z 385.88,A -85,B 0,C 180,E1 -24616.972,E2 -24616.972} C_VEL
LIN {X 0,Y 170.912,Z 374.501,A -85,B 0,C 180,E1 -24618.663,E2 -24618.663} C_VEL
LIN {X 0,Y 175.008,Z 359.741,A -85,B 0,C 180,E1 -24620.404,E2 -24620.404} C_VEL
LIN {X 0,Y 178.414,Z 344.956,A -85,B 0,C 180,E1 -24621.643,E2 -24621.643} C_VEL
LIN {X 0,Y 180.897,Z 329.701,A -85,B 0,C 180,E1 -24622.564,E2 -24622.564} C_VEL
LIN {X 0,Y 182.558,Z 312.42,A -85,B 0,C 180,E1 -24623.249,E2 -24623.249} C_VEL
LIN {X 0,Y 187.336,Z 250.052,A -85,B 0,C 180,E1 -24625.253,E2 -24625.253} C_VEL
LIN {X 0,Y 182.66,Z 237.3,A -85,B 0,C 180,E1 -24627.638,E2 -24627.638} C_VEL
LIN {X 0,Y 177.543,Z 225.021,A -85,B 0,C 180,E1 -24630.435,E2 -24630.435} C_VEL
LIN {X 0,Y 174.791,Z 219.705,A -85,B 0,C 180,E1 -24631.997,E2 -24631.997} C_VEL
LIN {X 0,Y 168.356,Z 209.279,A -85,B 0,C 180,E1 -24635.963,E2 -24635.963} C_VEL
LIN {X 0,Y 162.629,Z 200.974,A -85,B 0,C 180,E1 -24640.057,E2 -24640.057} C_VEL
LIN {X 0,Y 159.697,Z 196.871,A -85,B 0,C 180,E1 -24642.465,E2 -24642.465} C_VEL
LIN {X 0,Y 156.703,Z 193.033,A -85,B 0,C 180,E1 -24645.223,E2 -24645.223} C_VEL
LIN {X 0,Y 155.81,Z 191.827,A -85,B 0,C 180,E1 -24646.137,E2 -24646.137} C_VEL
LIN {X 0,Y 153.236,Z 188.918,A -85,B 0,C 180,E1 -24648.98,E2 -24648.98} C_VEL
LIN {X 0,Y 151.988,Z 186.632,A -85,B 0,C 180,E1 -24650.687,E2 -24650.687} C_VEL
LIN {X 0,Y 149.191,Z 184.047,A -85,B 0,C 180,E1 -24654.764,E2 -24654.764} C_VEL
LIN {X 0,Y 147.827,Z 181.083,A -85,B 0,C 180,E1 -24657.651,E2 -24657.651} C_VEL
LIN {X 0,Y 145.828,Z 180.108,A -85,B 0,C 180,E1 -24662.764,E2 -24662.764} C_VEL
LIN {X 0,Y 144.94,Z 179.527,A -85,B 0,C 180,E1 -24668.365,E2 -24668.365} C_VEL
LIN {X 0,Y 145.2,Z 180.089,A -85,B 0,C 180,E1 -24674.006,E2 -24674.006} C_VEL
LIN {X 0,Y 147.645,Z 181.491,A -85,B 0,C 180,E1 -24681.588,E2 -24681.588} C_VEL
LIN {X 0,Y 148.9,Z 184.257,A -85,B 0,C 180,E1 -24684.325,E2 -24684.325} C_VEL
LIN {X 0,Y 151.686,Z 186.729,A -85,B 0,C 180,E1 -24688.449,E2 -24688.449} C_VEL
LIN {X 0,Y 152.17,Z 187.212,A -85,B 0,C 180,E1 -24689.086,E2 -24689.086} C_VEL
LIN {X 0,Y 154.081,Z 190.354,A -85,B 0,C 180,E1 -24691.547,E2 -24691.547} C_VEL
LIN {X 0,Y 156.242,Z 192.503,A -85,B 0,C 180,E1 -24693.801,E2 -24693.801} C_VEL
LIN {X 0,Y 158.939,Z 196.235,A -85,B 0,C 180,E1 -24696.39,E2 -24696.39} C_VEL
LIN {X 0,Y 160.219,Z 197.945,A -85,B 0,C 180,E1 -24697.503,E2 -24697.503} C_VEL
LIN {X 0,Y 163.914,Z 203.007,A -85,B 0,C 180,E1 -24700.42,E2 -24700.42} C_VEL
LIN {X 0,Y 166.911,Z 207.332,A -85,B 0,C 180,E1 -24702.547,E2 -24702.547} C_VEL
LIN {X 0,Y 172.569,Z 216.056,A -85,B 0,C 180,E1 -24706.183,E2 -24706.183} C_VEL
LIN {X 0,Y 178.253,Z 225.826,A -85,B 0,C 180,E1 -24709.39,E2 -24709.39} C_VEL
LIN {X 0,Y 183.75,Z 236.496,A -85,B 0,C 180,E1 -24712.188,E2 -24712.188} C_VEL
LIN {X 0,Y 187.645,Z 244.7,A -85,B 0,C 180,E1 -24714.023,E2 -24714.023} C_VEL
LIN {X 0,Y 181.782,Z 318.018,A -85,B 0,C 180,E1 -24716.39,E2 -24716.39} C_VEL
LIN {X 0,Y 179.527,Z 333.885,A -85,B 0,C 180,E1 -24717.266,E2 -24717.266} C_VEL
LIN {X 0,Y 176.517,Z 348.955,A -85,B 0,C 180,E1 -24718.494,E2 -24718.494} C_VEL
LIN {X 0,Y 172.758,Z 363.518,A -85,B 0,C 180,E1 -24720.108,E2 -24720.108} C_VEL
LIN {X 0,Y 168.617,Z 376.816,A -85,B 0,C 180,E1 -24722.036,E2 -24722.036} C_VEL
LIN {X 0,Y 163.685,Z 390.35,A -85,B 0,C 180,E1 -24724.572,E2 -24724.572} C_VEL
LIN {X 0,Y 158.531,Z 402.675,A -85,B 0,C 180,E1 -24727.519,E2 -24727.519} C_VEL
LIN {X 0,Y 153.013,Z 414.729,A -85,B 0,C 180,E1 -24731.244,E2 -24731.244} C_VEL
LIN {X 0,Y 148.443,Z 424.113,A -85,B 0,C 180,E1 -24734.905,E2 -24734.905} C_VEL
LIN {X 0,Y 143.982,Z 433.22,A -85,B 0,C 180,E1 -24739.425,E2 -24739.425} C_VEL
LIN {X 0,Y 140.132,Z 440.886,A -85,B 0,C 180,E1 -24744.242,E2 -24744.242} C_VEL
LIN {X 0,Y 136.842,Z 448.008,A -85,B 0,C 180,E1 -24749.999,E2 -24749.999} C_VEL
LIN {X 0,Y 134.685,Z 453.601,A -85,B 0,C 180,E1 -24755.989,E2 -24755.989} C_VEL
LIN {X 0,Y 133.326,Z 457.836,A -85,B 0,C 180,E1 -24762.171,E2 -24762.171} C_VEL
LIN {X 0,Y 132.93,Z 460.78,A -85,B 0,C 180,E1 -24768.494,E2 -24768.494} C_VEL
LIN {X 0,Y 133.348,Z 462.48,A -85,B 0,C 180,E1 -24774.936,E2 -24774.936} C_VEL
LIN {X 0,Y 134.809,Z 462.914,A -85,B 0,C 180,E1 -24781.42,E2 -24781.42} C_VEL
LIN {X 0,Y 137.568,Z 462.054,A -85,B 0,C 180,E1 -24787.809,E2 -24787.809} C_VEL
LIN {X 0,Y 141.8,Z 459.856,A -85,B 0,C 180,E1 -24793.937,E2 -24793.937} C_VEL
LIN {X 0,Y 147.356,Z 456.246,A -85,B 0,C 180,E1 -24799.737,E2 -24799.737} C_VEL
LIN {X 0,Y 154.281,Z 451.125,A -85,B 0,C 180,E1 -24805.079,E2 -24805.079} C_VEL
LIN {X 0,Y 160.378,Z 446.156,A -85,B 0,C 180,E1 -24808.819,E2 -24808.819} C_VEL
LIN {X 0,Y 167.635,Z 439.555,A -85,B 0,C 180,E1 -24812.536,E2 -24812.536} C_VEL
LIN {X 0,Y 175.291,Z 431.873,A -85,B 0,C 180,E1 -24815.799,E2 -24815.799} C_VEL
LIN {X 0,Y 182.98,Z 423.205,A -85,B 0,C 180,E1 -24818.653,E2 -24818.653} C_VEL
LIN {X 0,Y 191.23,Z 412.698,A -85,B 0,C 180,E1 -24821.301,E2 -24821.301} C_VEL
LIN {X 0,Y 198.859,Z 401.613,A -85,B 0,C 180,E1 -24823.437,E2 -24823.437} C_VEL
LIN {X 0,Y 206.169,Z 389.254,A -85,B 0,C 180,E1 -24825.297,E2 -24825.297} C_VEL
LIN {X 0,Y 212.224,Z 377.256,A -85,B 0,C 180,E1 -24826.727,E2 -24826.727} C_VEL
LIN {X 0,Y 218.222,Z 363.013,A -85,B 0,C 180,E1 -24828.025,E2 -24828.025} C_VEL
LIN {X 0,Y 223.193,Z 348.117,A -85,B 0,C 180,E1 -24829.063,E2 -24829.063} C_VEL
LIN {X 0,Y 227.14,Z 332.62,A -85,B 0,C 180,E1 -24829.812,E2 -24829.812} C_VEL
LIN {X 0,Y 229.788,Z 317.377,A -85,B 0,C 180,E1 -24830.331,E2 -24830.331} C_VEL
LIN {X 0,Y 233.881,Z 277.838,A -85,B 0,C 180,E1 -24831.298,E2 -24831.298} C_VEL
LIN {X 0,Y 231.059,Z 271.837,A -85,B 0,C 180,E1 -24834.1,E2 -24834.1} C_VEL
LIN {X 0,Y 228.291,Z 266.217,A -85,B 0,C 180,E1 -24837.463,E2 -24837.463} C_VEL
LIN {X 0,Y 227.079,Z 263.934,A -85,B 0,C 180,E1 -24839.257,E2 -24839.257} C_VEL
LIN {X 0,Y 225.37,Z 260.29,A -85,B 0,C 180,E1 -24842.903,E2 -24842.903} C_VEL
LIN {X 0,Y 224.103,Z 258.824,A -85,B 0,C 180,E1 -24847.802,E2 -24847.802} C_VEL
LIN {X 0,Y 224.043,Z 258.871,A -85,B 0,C 180,E1 -24850.327,E2 -24850.327} C_VEL
LIN {X 0,Y 225.239,Z 260.408,A -85,B 0,C 180,E1 -24855.504,E2 -24855.504} C_VEL
LIN {X 0,Y 227.133,Z 264.524,A -85,B 0,C 180,E1 -24859.57,E2 -24859.57} C_VEL
LIN {X 0,Y 229.061,Z 269.272,A -85,B 0,C 180,E1 -24862.412,E2 -24862.412} C_VEL
LIN {X 0,Y 230.748,Z 273.567,A -85,B 0,C 180,E1 -24864.486,E2 -24864.486} C_VEL
LIN {X 0,Y 233.153,Z 280.142,A -85,B 0,C 180,E1 -24867.063,E2 -24867.063} C_VEL
LIN {X 0,Y 233.558,Z 281.403,A -85,B 0,C 180,E1 -24867.474,E2 -24867.474} C_VEL
LIN {X 0,Y 229.081,Z 324.224,A -85,B 0,C 180,E1 -24868.547,E2 -24868.547} C_VEL
LIN {X 0,Y 226.038,Z 340.122,A -85,B 0,C 180,E1 -24869.082,E2 -24869.082} C_VEL
LIN {X 0,Y 222.112,Z 354.537,A -85,B 0,C 180,E1 -24869.754,E2 -24869.754} C_VEL
LIN {X 0,Y 217.385,Z 367.992,A -85,B 0,C 180,E1 -24870.597,E2 -24870.597} C_VEL
LIN {X 0,Y 211.002,Z 382.789,A -85,B 0,C 180,E1 -24871.86,E2 -24871.86} C_VEL
LIN {X 0,Y 204.068,Z 396.083,A -85,B 0,C 180,E1 -24873.369,E2 -24873.369} C_VEL
LIN {X 0,Y 198.463,Z 405.377,A -85,B 0,C 180,E1 -24874.718,E2 -24874.718} C_VEL
LIN {X 0,Y 190.892,Z 416.645,A -85,B 0,C 180,E1 -24876.798,E2 -24876.798} C_VEL
LIN {X 0,Y 182.073,Z 427.937,A -85,B 0,C 180,E1 -24879.467,E2 -24879.467} C_VEL
LIN {X 0,Y 173.779,Z 437.339,A -85,B 0,C 180,E1 -24882.434,E2 -24882.434} C_VEL
LIN {X 0,Y 166.104,Z 445.103,A -85,B 0,C 180,E1 -24885.622,E2 -24885.622} C_VEL
LIN {X 0,Y 162.544,Z 448.077,A -85,B 0,C 180,E1 -24886.929,E2 -24886.929} C_VEL
LIN {X 0,Y 155.464,Z 452.567,A -85,B 0,C 180,E1 -24888.85,E2 -24888.85} C_VEL
LIN {X 0,Y 148.488,Z 456.55,A -85,B 0,C 180,E1 -24891.027,E2 -24891.027} C_VEL
LIN {X 0,Y 145.175,Z 458.681,A -85,B 0,C 180,E1 -24892.731,E2 -24892.731} C_VEL
LIN {X 0,Y 140.287,Z 462.2,A -85,B 0,C 180,E1 -24896.561,E2 -24896.561} C_VEL
LIN {X 0,Y 134.775,Z 465.805,A -85,B 0,C 180,E1 -24902.011,E2 -24902.011} C_VEL
LIN {X 0,Y 130.646,Z 468.267,A -85,B 0,C 180,E1 -24907.881,E2 -24907.881} C_VEL
LIN {X 0,Y 127.901,Z 469.609,A -85,B 0,C 180,E1 -24914.055,E2 -24914.055} C_VEL
LIN {X 0,Y 126.553,Z 469.818,A -85,B 0,C 180,E1 -24920.411,E2 -24920.411} C_VEL
LIN {X 0,Y 126.292,Z 468.936,A -85,B 0,C 180,E1 -24926.811,E2 -24926.811} C_VEL
LIN {X 0,Y 126.502,Z 468.073,A -85,B 0,C 180,E1 -24930.001,E2 -24930.001} C_VEL
LIN {X 0,Y 126.384,Z 465.386,A -85,B 0,C 180,E1 -24936.387,E2 -24936.387} C_VEL
LIN {X 0,Y 127.035,Z 461.392,A -85,B 0,C 180,E1 -24942.786,E2 -24942.786} C_VEL
LIN {X 0,Y 128.836,Z 455.98,A -85,B 0,C 180,E1 -24949.106,E2 -24949.106} C_VEL
LIN {X 0,Y 131.905,Z 449.033,A -85,B 0,C 180,E1 -24955.231,E2 -24955.231} C_VEL
LIN {X 0,Y 135.641,Z 441.501,A -85,B 0,C 180,E1 -24960.345,E2 -24960.345} C_VEL
LIN {X 0,Y 140.427,Z 432.445,A -85,B 0,C 180,E1 -24965.139,E2 -24965.139} C_VEL
LIN {X 0,Y 145.047,Z 423.147,A -85,B 0,C 180,E1 -24969.044,E2 -24969.044} C_VEL
LIN {X 0,Y 150.463,Z 412.19,A -85,B 0,C 180,E1 -24972.633,E2 -24972.633} C_VEL
LIN {X 0,Y 155.784,Z 400.165,A -85,B 0,C 180,E1 -24975.742,E2 -24975.742} C_VEL
LIN {X 0,Y 160.614,Z 388.497,A -85,B 0,C 180,E1 -24978.064,E2 -24978.064} C_VEL
LIN {X 0,Y 165.084,Z 376.093,A -85,B 0,C 180,E1 -24980.025,E2 -24980.025} C_VEL
LIN {X 0,Y 169.182,Z 362.241,A -85,B 0,C 180,E1 -24981.75,E2 -24981.75} C_VEL
LIN {X 0,Y 172.978,Z 346.788,A -85,B 0,C 180,E1 -24983.122,E2 -24983.122} C_VEL
LIN {X 0,Y 175.68,Z 331.342,A -85,B 0,C 180,E1 -24984.107,E2 -24984.107} C_VEL
LIN {X 0,Y 177.451,Z 315.12,A -85,B 0,C 180,E1 -24984.773,E2 -24984.773} C_VEL
LIN {X 0,Y 182.464,Z 252.504,A -85,B 0,C 180,E1 -24986.783,E2 -24986.783} C_VEL
LIN {X 0,Y 178.841,Z 242.094,A -85,B 0,C 180,E1 -24988.787,E2 -24988.787} C_VEL
LIN {X 0,Y 173.734,Z 229.396,A -85,B 0,C 180,E1 -24991.785,E2 -24991.785} C_VEL
LIN {X 0,Y 170.903,Z 223.935,A -85,B 0,C 180,E1 -24993.508,E2 -24993.508} C_VEL
LIN {X 0,Y 165.463,Z 214.884,A -85,B 0,C 180,E1 -24997.114,E2 -24997.114} C_VEL
LIN {X 0,Y 160.205,Z 207.038,A -85,B 0,C 180,E1 -25001.083,E2 -25001.083} C_VEL
LIN {X 0,Y 156.922,Z 202.472,A -85,B 0,C 180,E1 -25003.967,E2 -25003.967} C_VEL
LIN {X 0,Y 153.993,Z 198.35,A -85,B 0,C 180,E1 -25006.968,E2 -25006.968} C_VEL
LIN {X 0,Y 151.393,Z 195.147,A -85,B 0,C 180,E1 -25010.06,E2 -25010.06} C_VEL
LIN {X 0,Y 150.572,Z 193.474,A -85,B 0,C 180,E1 -25011.276,E2 -25011.276} C_VEL
LIN {X 0,Y 147.815,Z 190.735,A -85,B 0,C 180,E1 -25015.516,E2 -25015.516} C_VEL
LIN {X 0,Y 146.604,Z 187.995,A -85,B 0,C 180,E1 -25018.266,E2 -25018.266} C_VEL
LIN {X 0,Y 144.564,Z 187.029,A -85,B 0,C 180,E1 -25024.183,E2 -25024.183} C_VEL
LIN {X 0,Y 144.045,Z 186.551,A -85,B 0,C 180,E1 -25028.418,E2 -25028.418} C_VEL
LIN {X 0,Y 144.463,Z 187.298,A -85,B 0,C 180,E1 -25034.977,E2 -25034.977} C_VEL
LIN {X 0,Y 146.415,Z 188.459,A -85,B 0,C 180,E1 -25040.956,E2 -25040.956} C_VEL
LIN {X 0,Y 147.949,Z 191.472,A -85,B 0,C 180,E1 -25044.328,E2 -25044.328} C_VEL
LIN {X 0,Y 150.617,Z 193.966,A -85,B 0,C 180,E1 -25048.331,E2 -25048.331} C_VEL
LIN {X 0,Y 152.895,Z 197.462,A -85,B 0,C 180,E1 -25051.333,E2 -25051.333} C_VEL
LIN {X 0,Y 154.444,Z 199.121,A -85,B 0,C 180,E1 -25053.023,E2 -25053.023} C_VEL
LIN {X 0,Y 157.291,Z 203.021,A -85,B 0,C 180,E1 -25055.862,E2 -25055.862} C_VEL
LIN {X 0,Y 161.722,Z 209.431,A -85,B 0,C 180,E1 -25059.632,E2 -25059.632} C_VEL
LIN {X 0,Y 165.99,Z 215.84,A -85,B 0,C 180,E1 -25062.742,E2 -25062.742} C_VEL
LIN {X 0,Y 171.663,Z 225.246,A -85,B 0,C 180,E1 -25066.43,E2 -25066.43} C_VEL
LIN {X 0,Y 178.084,Z 237.387,A -85,B 0,C 180,E1 -25070.083,E2 -25070.083} C_VEL
LIN {X 0,Y 182.622,Z 247.109,A -85,B 0,C 180,E1 -25072.425,E2 -25072.425} C_VEL
LIN {X 0,Y 179.322,Z 288.954,A -85,B 0,C 180,E1 -25073.783,E2 -25073.783} C_VEL
LIN {X 0,Y 176.771,Z 318.676,A -85,B 0,C 180,E1 -25074.795,E2 -25074.795} C_VEL
LIN {X 0,Y 174.445,Z 334.296,A -85,B 0,C 180,E1 -25075.664,E2 -25075.664} C_VEL
LIN {X 0,Y 171.354,Z 349.295,A -85,B 0,C 180,E1 -25076.905,E2 -25076.905} C_VEL
LIN {X 0,Y 167.736,Z 362.933,A -85,B 0,C 180,E1 -25078.415,E2 -25078.415} C_VEL
LIN {X 0,Y 163.419,Z 376.362,A -85,B 0,C 180,E1 -25080.357,E2 -25080.357} C_VEL
LIN {X 0,Y 158.576,Z 389.314,A -85,B 0,C 180,E1 -25082.778,E2 -25082.778} C_VEL
LIN {X 0,Y 152.911,Z 402.456,A -85,B 0,C 180,E1 -25085.925,E2 -25085.925} C_VEL
LIN {X 0,Y 147.1,Z 414.597,A -85,B 0,C 180,E1 -25089.733,E2 -25089.733} C_VEL
LIN {X 0,Y 142.28,Z 424.027,A -85,B 0,C 180,E1 -25093.498,E2 -25093.498} C_VEL
LIN {X 0,Y 137.528,Z 433.229,A -85,B 0,C 180,E1 -25098.204,E2 -25098.204} C_VEL
LIN {X 0,Y 133.489,Z 440.891,A -85,B 0,C 180,E1 -25103.196,E2 -25103.196} C_VEL
LIN {X 0,Y 130.35,Z 447.228,A -85,B 0,C 180,E1 -25108.454,E2 -25108.454} C_VEL
LIN {X 0,Y 127.923,Z 453.04,A -85,B 0,C 180,E1 -25114.726,E2 -25114.726} C_VEL
LIN {X 0,Y 126.623,Z 456.536,A -85,B 0,C 180,E1 -25119.584,E2 -25119.584} C_VEL
LIN {X 0,Y 125.881,Z 459.978,A -85,B 0,C 180,E1 -25126.208,E2 -25126.208} C_VEL
LIN {X 0,Y 125.996,Z 462.168,A -85,B 0,C 180,E1 -25132.982,E2 -25132.982} C_VEL
LIN {X 0,Y 126.668,Z 462.949,A -85,B 0,C 180,E1 -25137.406,E2 -25137.406} C_VEL
LIN {X 0,Y 129.097,Z 462.946,A -85,B 0,C 180,E1 -25145.252,E2 -25145.252} C_VEL
LIN {X 0,Y 133.163,Z 461.369,A -85,B 0,C 180,E1 -25152.362,E2 -25152.362} C_VEL
LIN {X 0,Y 138.636,Z 458.368,A -85,B 0,C 180,E1 -25158.773,E2 -25158.773} C_VEL
LIN {X 0,Y 145.576,Z 453.864,A -85,B 0,C 180,E1 -25164.595,E2 -25164.595} C_VEL
LIN {X 0,Y 151.832,Z 449.325,A -85,B 0,C 180,E1 -25168.693,E2 -25168.693} C_VEL
LIN {X 0,Y 158.608,Z 443.771,A -85,B 0,C 180,E1 -25172.399,E2 -25172.399} C_VEL
LIN {X 0,Y 167.078,Z 436.12,A -85,B 0,C 180,E1 -25176.189,E2 -25176.189} C_VEL
LIN {X 0,Y 176.227,Z 426.771,A -85,B 0,C 180,E1 -25179.583,E2 -25179.583} C_VEL
LIN {X 0,Y 184.552,Z 417.011,A -85,B 0,C 180,E1 -25182.262,E2 -25182.262} C_VEL
LIN {X 0,Y 192.405,Z 406.566,A -85,B 0,C 180,E1 -25184.449,E2 -25184.449} C_VEL
LIN {X 0,Y 199.586,Z 395.6,A -85,B 0,C 180,E1 -25186.271,E2 -25186.271} C_VEL
LIN {X 0,Y 206.64,Z 383.041,A -85,B 0,C 180,E1 -25187.905,E2 -25187.905} C_VEL
LIN {X 0,Y 212.838,Z 369.953,A -85,B 0,C 180,E1 -25189.215,E2 -25189.215} C_VEL
LIN {X 0,Y 218.34,Z 355.653,A -85,B 0,C 180,E1 -25190.319,E2 -25190.319} C_VEL
LIN {X 0,Y 222.3,Z 342.774,A -85,B 0,C 180,E1 -25191.064,E2 -25191.064} C_VEL
LIN {X 0,Y 225.966,Z 326.795,A -85,B 0,C 180,E1 -25191.726,E2 -25191.726} C_VEL
LIN {X 0,Y 228.326,Z 310.184,A -85,B 0,C 180,E1 -25192.19,E2 -25192.19} C_VEL
LIN {X 0,Y 231.23,Z 282.06,A -85,B 0,C 180,E1 -25192.852,E2 -25192.852} C_VEL
LIN {X 0,Y 228.432,Z 276.021,A -85,B 0,C 180,E1 -25195.99,E2 -25195.99} C_VEL
LIN {X 0,Y 226.469,Z 271.878,A -85,B 0,C 180,E1 -25198.72,E2 -25198.72} C_VEL
LIN {X 0,Y 225.711,Z 270.489,A -85,B 0,C 180,E1 -25199.999,E2 -25199.999} C_VEL
LIN {X 0,Y 224.214,Z 266.929,A -85,B 0,C 180,E1 -25203.594,E2 -25203.594} C_VEL
LIN {X 0,Y 223.12,Z 265.701,A -85,B 0,C 180,E1 -25209.061,E2 -25209.061} C_VEL
LIN {X 0,Y 224.213,Z 267.356,A -85,B 0,C 180,E1 -25215.194,E2 -25215.194} C_VEL
LIN {X 0,Y 225.872,Z 271.192,A -85,B 0,C 180,E1 -25219.034,E2 -25219.034} C_VEL
LIN {X 0,Y 227.744,Z 276.178,A -85,B 0,C 180,E1 -25221.995,E2 -25221.995} C_VEL
LIN {X 0,Y 229.478,Z 280.854,A -85,B 0,C 180,E1 -25224.223,E2 -25224.223} C_VEL
LIN {X 0,Y 230.947,Z 285.124,A -85,B 0,C 180,E1 -25225.906,E2 -25225.906} C_VEL
LIN {X 0,Y 226.731,Z 324.092,A -85,B 0,C 180,E1 -25226.861,E2 -25226.861} C_VEL
LIN {X 0,Y 223.697,Z 339.724,A -85,B 0,C 180,E1 -25227.376,E2 -25227.376} C_VEL
LIN {X 0,Y 219.479,Z 354.771,A -85,B 0,C 180,E1 -25228.045,E2 -25228.045} C_VEL
LIN {X 0,Y 214.653,Z 368.169,A -85,B 0,C 180,E1 -25228.858,E2 -25228.858} C_VEL
LIN {X 0,Y 208.117,Z 382.84,A -85,B 0,C 180,E1 -25230.079,E2 -25230.079} C_VEL
LIN {X 0,Y 201.007,Z 396.055,A -85,B 0,C 180,E1 -25231.545,E2 -25231.545} C_VEL
LIN {X 0,Y 194.564,Z 406.337,A -85,B 0,C 180,E1 -25233.014,E2 -25233.014} C_VEL
LIN {X 0,Y 186.755,Z 417.417,A -85,B 0,C 180,E1 -25235.066,E2 -25235.066} C_VEL
LIN {X 0,Y 177.67,Z 428.549,A -85,B 0,C 180,E1 -25237.71,E2 -25237.71} C_VEL
LIN {X 0,Y 169.08,Z 437.814,A -85,B 0,C 180,E1 -25240.662,E2 -25240.662} C_VEL
LIN {X 0,Y 160.778,Z 445.744,A -85,B 0,C 180,E1 -25243.992,E2 -25243.992} C_VEL
LIN {X 0,Y 154.543,Z 451.218,A -85,B 0,C 180,E1 -25246.99,E2 -25246.99} C_VEL
LIN {X 0,Y 146.922,Z 457.377,A -85,B 0,C 180,E1 -25251.549,E2 -25251.549} C_VEL
LIN {X 0,Y 145.175,Z 458.681,A -85,B 0,C 180,E1 -25252.731,E2 -25252.731} C_VEL
LIN {X 0,Y 141.923,Z 460.676,A -85,B 0,C 180,E1 -25254.54,E2 -25254.54} C_VEL
LIN {X 0,Y 135.276,Z 463.54,A -85,B 0,C 180,E1 -25257.361,E2 -25257.361} C_VEL
LIN {X 0,Y 129.012,Z 465.819,A -85,B 0,C 180,E1 -25260.546,E2 -25260.546} C_VEL
LIN {X 0,Y 126.467,Z 466.895,A -85,B 0,C 180,E1 -25262.884,E2 -25262.884} C_VEL
LIN {X 0,Y 122.384,Z 468.953,A -85,B 0,C 180,E1 -25269.847,E2 -25269.847} C_VEL
LIN {X 0,Y 120.115,Z 469.67,A -85,B 0,C 180,E1 -25276.466,E2 -25276.466} C_VEL
LIN {X 0,Y 119.212,Z 469.248,A -85,B 0,C 180,E1 -25283.23,E2 -25283.23} C_VEL
LIN {X 0,Y 119.414,Z 467.719,A -85,B 0,C 180,E1 -25290.001,E2 -25290.001} C_VEL
LIN {X 0,Y 119.275,Z 466.486,A -85,B 0,C 180,E1 -25293.379,E2 -25293.379} C_VEL
LIN {X 0,Y 119.57,Z 463.068,A -85,B 0,C 180,E1 -25300.158,E2 -25300.158} C_VEL
LIN {X 0,Y 120.854,Z 458.288,A -85,B 0,C 180,E1 -25306.905,E2 -25306.905} C_VEL
LIN {X 0,Y 123.56,Z 452.028,A -85,B 0,C 180,E1 -25313.464,E2 -25313.464} C_VEL
LIN {X 0,Y 127.612,Z 444.102,A -85,B 0,C 180,E1 -25319.715,E2 -25319.715} C_VEL
LIN {X 0,Y 132.317,Z 435.64,A -85,B 0,C 180,E1 -25324.821,E2 -25324.821} C_VEL
LIN {X 0,Y 137.778,Z 425.445,A -85,B 0,C 180,E1 -25329.575,E2 -25329.575} C_VEL
LIN {X 0,Y 143.296,Z 414.876,A -85,B 0,C 180,E1 -25333.366,E2 -25333.366} C_VEL
LIN {X 0,Y 148.759,Z 403.407,A -85,B 0,C 180,E1 -25336.585,E2 -25336.585} C_VEL
LIN {X 0,Y 154.205,Z 390.968,A -85,B 0,C 180,E1 -25339.263,E2 -25339.263} C_VEL
LIN {X 0,Y 159.39,Z 377.406,A -85,B 0,C 180,E1 -25341.506,E2 -25341.506} C_VEL
LIN {X 0,Y 163.625,Z 363.792,A -85,B 0,C 180,E1 -25343.27,E2 -25343.27} C_VEL
LIN {X 0,Y 167.513,Z 349.062,A -85,B 0,C 180,E1 -25344.639,E2 -25344.639} C_VEL
LIN {X 0,Y 170.405,Z 333.763,A -85,B 0,C 180,E1 -25345.695,E2 -25345.695} C_VEL
LIN {X 0,Y 172.281,Z 319.561,A -85,B 0,C 180,E1 -25346.316,E2 -25346.316} C_VEL
LIN {X 0,Y 177.62,Z 254.229,A -85,B 0,C 180,E1 -25348.484,E2 -25348.484} C_VEL
LIN {X 0,Y 173.14,Z 241.691,A -85,B 0,C 180,E1 -25351.183,E2 -25351.183} C_VEL
LIN {X 0,Y 169.438,Z 232.404,A -85,B 0,C 180,E1 -25353.585,E2 -25353.585} C_VEL
LIN {X 0,Y 164.162,Z 222.984,A -85,B 0,C 180,E1 -25357.172,E2 -25357.172} C_VEL
LIN {X 0,Y 159.554,Z 215.806,A -85,B 0,C 180,E1 -25360.668,E2 -25360.668} C_VEL
LIN {X 0,Y 157.168,Z 212.233,A -85,B 0,C 180,E1 -25362.721,E2 -25362.721} C_VEL
LIN {X 0,Y 154.761,Z 208.601,A -85,B 0,C 180,E1 -25365.033,E2 -25365.033} C_VEL
LIN {X 0,Y 152.092,Z 204.761,A -85,B 0,C 180,E1 -25367.952,E2 -25367.952} C_VEL
LIN {X 0,Y 149.625,Z 201.417,A -85,B 0,C 180,E1 -25371.135,E2 -25371.135} C_VEL
LIN {X 0,Y 148.988,Z 200.108,A -85,B 0,C 180,E1 -25372.147,E2 -25372.147} C_VEL
LIN {X 0,Y 146.266,Z 197.092,A -85,B 0,C 180,E1 -25376.691,E2 -25376.691} C_VEL
LIN {X 0,Y 145.325,Z 194.826,A -85,B 0,C 180,E1 -25379.072,E2 -25379.072} C_VEL
LIN {X 0,Y 143.141,Z 193.597,A -85,B 0,C 180,E1 -25388.471,E2 -25388.471} C_VEL
LIN {X 0,Y 143.768,Z 194.5,A -85,B 0,C 180,E1 -25395.956,E2 -25395.956} C_VEL
LIN {X 0,Y 145.23,Z 195.413,A -85,B 0,C 180,E1 -25400.37,E2 -25400.37} C_VEL
LIN {X 0,Y 146.806,Z 198.473,A -85,B 0,C 180,E1 -25403.989,E2 -25403.989} C_VEL
LIN {X 0,Y 149.168,Z 200.814,A -85,B 0,C 180,E1 -25407.672,E2 -25407.672} C_VEL
LIN {X 0,Y 151.373,Z 204.193,A -85,B 0,C 180,E1 -25410.713,E2 -25410.713} C_VEL
LIN {X 0,Y 152.735,Z 205.829,A -85,B 0,C 180,E1 -25412.29,E2 -25412.29} C_VEL
LIN {X 0,Y 156.014,Z 210.632,A -85,B 0,C 180,E1 -25415.699,E2 -25415.699} C_VEL
LIN {X 0,Y 160.515,Z 217.188,A -85,B 0,C 180,E1 -25419.58,E2 -25419.58} C_VEL
LIN {X 0,Y 166.531,Z 227.117,A -85,B 0,C 180,E1 -25423.976,E2 -25423.976} C_VEL
LIN {X 0,Y 171.541,Z 236.472,A -85,B 0,C 180,E1 -25427.195,E2 -25427.195} C_VEL
LIN {X 0,Y 176.377,Z 246.526,A -85,B 0,C 180,E1 -25429.993,E2 -25429.993} C_VEL
LIN {X 0,Y 177.866,Z 249.862,A -85,B 0,C 180,E1 -25430.807,E2 -25430.807} C_VEL
LIN {X 0,Y 172.057,Z 318.051,A -85,B 0,C 180,E1 -25433.042,E2 -25433.042} C_VEL
LIN {X 0,Y 169.686,Z 333.925,A -85,B 0,C 180,E1 -25433.919,E2 -25433.919} C_VEL
LIN {X 0,Y 166.313,Z 349.647,A -85,B 0,C 180,E1 -25435.215,E2 -25435.215} C_VEL
LIN {X 0,Y 162.291,Z 364.138,A -85,B 0,C 180,E1 -25436.856,E2 -25436.856} C_VEL
LIN {X 0,Y 157.817,Z 377.409,A -85,B 0,C 180,E1 -25438.821,E2 -25438.821} C_VEL
LIN {X 0,Y 152.613,Z 390.637,A -85,B 0,C 180,E1 -25441.37,E2 -25441.37} C_VEL
LIN {X 0,Y 146.896,Z 403.219,A -85,B 0,C 180,E1 -25444.494,E2 -25444.494} C_VEL
LIN {X 0,Y 141.28,Z 414.441,A -85,B 0,C 180,E1 -25448.092,E2 -25448.092} C_VEL
LIN {X 0,Y 136.208,Z 423.901,A -85,B 0,C 180,E1 -25451.964,E2 -25451.964} C_VEL
LIN {X 0,Y 131.156,Z 433.161,A -85,B 0,C 180,E1 -25456.835,E2 -25456.835} C_VEL
LIN {X 0,Y 126.882,Z 440.867,A -85,B 0,C 180,E1 -25462.039,E2 -25462.039} C_VEL
LIN {X 0,Y 123.145,Z 448.073,A -85,B 0,C 180,E1 -25468.364,E2 -25468.364} C_VEL
LIN {X 0,Y 120.711,Z 453.656,A -85,B 0,C 180,E1 -25474.896,E2 -25474.896} C_VEL
LIN {X 0,Y 119.382,Z 457.116,A -85,B 0,C 180,E1 -25480.171,E2 -25480.171} C_VEL
LIN {X 0,Y 118.77,Z 460.459,A -85,B 0,C 180,E1 -25487.208,E2 -25487.208} C_VEL
LIN {X 0,Y 119.037,Z 462.547,A -85,B 0,C 180,E1 -25494.41,E2 -25494.41} C_VEL
LIN {X 0,Y 119.72,Z 463.145,A -85,B 0,C 180,E1 -25498.288,E2 -25498.288} C_VEL
LIN {X 0,Y 121.85,Z 463.276,A -85,B 0,C 180,E1 -25505.223,E2 -25505.223} C_VEL
LIN {X 0,Y 125.617,Z 462.141,A -85,B 0,C 180,E1 -25512.172,E2 -25512.172} C_VEL
LIN {X 0,Y 130.927,Z 459.658,A -85,B 0,C 180,E1 -25518.719,E2 -25518.719} C_VEL
LIN {X 0,Y 137.736,Z 455.751,A -85,B 0,C 180,E1 -25524.724,E2 -25524.724} C_VEL
LIN {X 0,Y 145.869,Z 450.319,A -85,B 0,C 180,E1 -25530.138,E2 -25530.138} C_VEL
LIN {X 0,Y 152.727,Z 445.134,A -85,B 0,C 180,E1 -25533.807,E2 -25533.807} C_VEL
LIN {X 0,Y 161.474,Z 437.76,A -85,B 0,C 180,E1 -25537.649,E2 -25537.649} C_VEL
LIN {X 0,Y 170.89,Z 428.735,A -85,B 0,C 180,E1 -25541.064,E2 -25541.064} C_VEL
LIN {X 0,Y 179.051,Z 419.829,A -85,B 0,C 180,E1 -25543.636,E2 -25543.636} C_VEL
LIN {X 0,Y 186.716,Z 410.337,A -85,B 0,C 180,E1 -25545.747,E2 -25545.747} C_VEL
LIN {X 0,Y 195.058,Z 398.496,A -85,B 0,C 180,E1 -25547.771,E2 -25547.771} C_VEL
LIN {X 0,Y 202.623,Z 385.802,A -85,B 0,C 180,E1 -25549.473,E2 -25549.473} C_VEL
LIN {X 0,Y 209.138,Z 372.823,A -85,B 0,C 180,E1 -25550.796,E2 -25550.796} C_VEL
LIN {X 0,Y 214.612,Z 359.614,A -85,B 0,C 180,E1 -25551.833,E2 -25551.833} C_VEL
LIN {X 0,Y 218.942,Z 346.66,A -85,B 0,C 180,E1 -25552.622,E2 -25552.622} C_VEL
LIN {X 0,Y 222.902,Z 331.103,A -85,B 0,C 180,E1 -25553.308,E2 -25553.308} C_VEL
LIN {X 0,Y 225.54,Z 315.615,A -85,B 0,C 180,E1 -25553.778,E2 -25553.778} C_VEL
LIN {X 0,Y 228.683,Z 286.399,A -85,B 0,C 180,E1 -25554.488,E2 -25554.488} C_VEL
LIN {X 0,Y 226.613,Z 281.788,A -85,B 0,C 180,E1 -25557.077,E2 -25557.077} C_VEL
LIN {X 0,Y 224.948,Z 277.883,A -85,B 0,C 180,E1 -25559.717,E2 -25559.717} C_VEL
LIN {X 0,Y 223.155,Z 273.851,A -85,B 0,C 180,E1 -25564.024,E2 -25564.024} C_VEL
LIN {X 0,Y 222.22,Z 272.756,A -85,B 0,C 180,E1 -25569.098,E2 -25569.098} C_VEL
LIN {X 0,Y 223.205,Z 274.367,A -85,B 0,C 180,E1 -25574.926,E2 -25574.926} C_VEL
LIN {X 0,Y 224.675,Z 278.007,A -85,B 0,C 180,E1 -25578.569,E2 -25578.569} C_VEL
LIN {X 0,Y 226.324,Z 282.714,A -85,B 0,C 180,E1 -25581.397,E2 -25581.397} C_VEL
LIN {X 0,Y 228.319,Z 288.689,A -85,B 0,C 180,E1 -25584.115,E2 -25584.115} C_VEL
LIN {X 0,Y 228.449,Z 289.112,A -85,B 0,C 180,E1 -25584.279,E2 -25584.279} C_VEL
LIN {X 0,Y 224.565,Z 324.019,A -85,B 0,C 180,E1 -25585.138,E2 -25585.138} C_VEL
LIN {X 0,Y 221.453,Z 339.682,A -85,B 0,C 180,E1 -25585.639,E2 -25585.639} C_VEL
LIN {X 0,Y 217.049,Z 355.002,A -85,B 0,C 180,E1 -25586.297,E2 -25586.297} C_VEL
LIN {X 0,Y 211.382,Z 370.061,A -85,B 0,C 180,E1 -25587.206,E2 -25587.206} C_VEL
LIN {X 0,Y 205.447,Z 382.914,A -85,B 0,C 180,E1 -25588.254,E2 -25588.254} C_VEL
LIN {X 0,Y 198.151,Z 396.088,A -85,B 0,C 180,E1 -25589.663,E2 -25589.663} C_VEL
LIN {X 0,Y 190.829,Z 407.402,A -85,B 0,C 180,E1 -25591.246,E2 -25591.246} C_VEL
LIN {X 0,Y 181.476,Z 419.963,A -85,B 0,C 180,E1 -25593.632,E2 -25593.632} C_VEL
LIN {X 0,Y 172.121,Z 430.603,A -85,B 0,C 180,E1 -25596.253,E2 -25596.253} C_VEL
LIN {X 0,Y 163.323,Z 439.502,A -85,B 0,C 180,E1 -25599.236,E2 -25599.236} C_VEL
LIN {X 0,Y 153.822,Z 447.919,A -85,B 0,C 180,E1 -25603.029,E2 -25603.029} C_VEL
LIN {X 0,Y 147.376,Z 453.112,A -85,B 0,C 180,E1 -25606.255,E2 -25606.255} C_VEL
LIN {X 0,Y 139.153,Z 459.108,A -85,B 0,C 180,E1 -25611.244,E2 -25611.244} C_VEL
LIN {X 0,Y 134.378,Z 462.295,A -85,B 0,C 180,E1 -25614.88,E2 -25614.88} C_VEL
LIN {X 0,Y 128.514,Z 465.805,A -85,B 0,C 180,E1 -25620.517,E2 -25620.517} C_VEL
LIN {X 0,Y 126.467,Z 466.895,A -85,B 0,C 180,E1 -25622.884,E2 -25622.884} C_VEL
LIN {X 0,Y 124.151,Z 467.846,A -85,B 0,C 180,E1 -25625.334,E2 -25625.334} C_VEL
LIN {X 0,Y 119.034,Z 468.893,A -85,B 0,C 180,E1 -25629.303,E2 -25629.303} C_VEL
LIN {X 0,Y 115.178,Z 469.366,A -85,B 0,C 180,E1 -25632.705,E2 -25632.705} C_VEL
LIN {X 0,Y 113.287,Z 469.479,A -85,B 0,C 180,E1 -25635.522,E2 -25635.522} C_VEL
LIN {X 0,Y 112.972,Z 469.451,A -85,B 0,C 180,E1 -25636.51,E2 -25636.51} C_VEL
LIN {X 0,Y 112.16,Z 468.982,A -85,B 0,C 180,E1 -25642.802,E2 -25642.802} C_VEL
LIN {X 0,Y 112.328,Z 467.364,A -85,B 0,C 180,E1 -25650.001,E2 -25650.001} C_VEL
LIN {X 0,Y 112.222,Z 464.491,A -85,B 0,C 180,E1 -25657.197,E2 -25657.197} C_VEL
LIN {X 0,Y 113.112,Z 460.308,A -85,B 0,C 180,E1 -25664.392,E2 -25664.392} C_VEL
LIN {X 0,Y 115.337,Z 454.702,A -85,B 0,C 180,E1 -25671.447,E2 -25671.447} C_VEL
LIN {X 0,Y 119.032,Z 447.521,A -85,B 0,C 180,E1 -25678.188,E2 -25678.188} C_VEL
LIN {X 0,Y 123.442,Z 439.806,A -85,B 0,C 180,E1 -25683.719,E2 -25683.719} C_VEL
LIN {X 0,Y 128.892,Z 430.484,A -85,B 0,C 180,E1 -25688.835,E2 -25688.835} C_VEL
LIN {X 0,Y 134.212,Z 420.926,A -85,B 0,C 180,E1 -25692.904,E2 -25692.904} C_VEL
LIN {X 0,Y 140.688,Z 408.56,A -85,B 0,C 180,E1 -25696.938,E2 -25696.938} C_VEL
LIN {X 0,Y 146.099,Z 397.13,A -85,B 0,C 180,E1 -25699.79,E2 -25699.79} C_VEL
LIN {X 0,Y 151.956,Z 383.435,A -85,B 0,C 180,E1 -25702.378,E2 -25702.378} C_VEL
LIN {X 0,Y 157.042,Z 369.199,A -85,B 0,C 180,E1 -25704.425,E2 -25704.425} C_VEL
LIN {X 0,Y 161.18,Z 355.073,A -85,B 0,C 180,E1 -25705.943,E2 -25705.943} C_VEL
LIN {X 0,Y 164.713,Z 339.555,A -85,B 0,C 180,E1 -25707.146,E2 -25707.146} C_VEL
LIN {X 0,Y 167.158,Z 324.175,A -85,B 0,C 180,E1 -25707.948,E2 -25707.948} C_VEL
LIN {X 0,Y 173.055,Z 256.648,A -85,B 0,C 180,E1 -25710.183,E2 -25710.183} C_VEL
LIN {X 0,Y 168.433,Z 243.299,A -85,B 0,C 180,E1 -25713.252,E2 -25713.252} C_VEL
LIN {X 0,Y 165.629,Z 236.407,A -85,B 0,C 180,E1 -25715.228,E2 -25715.228} C_VEL
LIN {X 0,Y 160.22,Z 226.672,A -85,B 0,C 180,E1 -25719.206,E2 -25719.206} C_VEL
LIN {X 0,Y 155.533,Z 219.17,A -85,B 0,C 180,E1 -25723.218,E2 -25723.218} C_VEL
LIN {X 0,Y 152.607,Z 214.677,A -85,B 0,C 180,E1 -25726.179,E2 -25726.179} C_VEL
LIN {X 0,Y 150.319,Z 211.213,A -85,B 0,C 180,E1 -25728.87,E2 -25728.87} C_VEL
LIN {X 0,Y 147.998,Z 207.866,A -85,B 0,C 180,E1 -25732.094,E2 -25732.094} C_VEL
LIN {X 0,Y 147.283,Z 206.661,A -85,B 0,C 180,E1 -25733.238,E2 -25733.238} C_VEL
LIN {X 0,Y 144.835,Z 203.5,A -85,B 0,C 180,E1 -25737.771,E2 -25737.771} C_VEL
LIN {X 0,Y 144.154,Z 201.72,A -85,B 0,C 180,E1 -25739.689,E2 -25739.689} C_VEL
LIN {X 0,Y 142.228,Z 200.648,A -85,B 0,C 180,E1 -25748.775,E2 -25748.775} C_VEL
LIN {X 0,Y 143.879,Z 202.098,A -85,B 0,C 180,E1 -25759.253,E2 -25759.253} C_VEL
LIN {X 0,Y 146.319,Z 206.212,A -85,B 0,C 180,E1 -25764.804,E2 -25764.804} C_VEL
LIN {X 0,Y 147.653,Z 207.488,A -85,B 0,C 180,E1 -25766.88,E2 -25766.88} C_VEL
LIN {X 0,Y 150.128,Z 211.23,A -85,B 0,C 180,E1 -25770.403,E2 -25770.403} C_VEL
LIN {X 0,Y 151.201,Z 212.803,A -85,B 0,C 180,E1 -25771.725,E2 -25771.725} C_VEL
LIN {X 0,Y 153.842,Z 216.767,A -85,B 0,C 180,E1 -25774.626,E2 -25774.626} C_VEL
LIN {X 0,Y 158.114,Z 223.276,A -85,B 0,C 180,E1 -25778.564,E2 -25778.564} C_VEL
LIN {X 0,Y 163.715,Z 232.81,A -85,B 0,C 180,E1 -25782.886,E2 -25782.886} C_VEL
LIN {X 0,Y 168.628,Z 242.454,A -85,B 0,C 180,E1 -25786.253,E2 -25786.253} C_VEL
LIN {X 0,Y 173.028,Z 252.05,A -85,B 0,C 180,E1 -25788.963,E2 -25788.963} C_VEL
LIN {X 0,Y 173.274,Z 252.78,A -85,B 0,C 180,E1 -25789.119,E2 -25789.119} C_VEL
LIN {X 0,Y 167.365,Z 318.59,A -85,B 0,C 180,E1 -25791.247,E2 -25791.247} C_VEL
LIN {X 0,Y 164.914,Z 334.333,A -85,B 0,C 180,E1 -25792.124,E2 -25792.124} C_VEL
LIN {X 0,Y 161.702,Z 348.884,A -85,B 0,C 180,E1 -25793.299,E2 -25793.299} C_VEL
LIN {X 0,Y 157.549,Z 363.572,A -85,B 0,C 180,E1 -25794.946,E2 -25794.946} C_VEL
LIN {X 0,Y 152.919,Z 376.956,A -85,B 0,C 180,E1 -25796.922,E2 -25796.922} C_VEL
LIN {X 0,Y 147.33,Z 390.636,A -85,B 0,C 180,E1 -25799.558,E2 -25799.558} C_VEL
LIN {X 0,Y 141.499,Z 402.988,A -85,B 0,C 180,E1 -25802.648,E2 -25802.648} C_VEL
LIN {X 0,Y 135.59,Z 414.278,A -85,B 0,C 180,E1 -25806.314,E2 -25806.314} C_VEL
LIN {X 0,Y 129.429,Z 425.223,A -85,B 0,C 180,E1 -25810.984,E2 -25810.984} C_VEL
LIN {X 0,Y 124.204,Z 434.305,A -85,B 0,C 180,E1 -25816.084,E2 -25816.084} C_VEL
LIN {X 0,Y 119.748,Z 441.874,A -85,B 0,C 180,E1 -25821.561,E2 -25821.561} C_VEL
LIN {X 0,Y 115.928,Z 448.92,A -85,B 0,C 180,E1 -25828.262,E2 -25828.262} C_VEL
LIN {X 0,Y 113.945,Z 453.164,A -85,B 0,C 180,E1 -25833.535,E2 -25833.535} C_VEL
LIN {X 0,Y 112.485,Z 456.703,A -85,B 0,C 180,E1 -25838.985,E2 -25838.985} C_VEL
LIN {X 0,Y 111.751,Z 459.45,A -85,B 0,C 180,E1 -25844.568,E2 -25844.568} C_VEL
LIN {X 0,Y 111.649,Z 461.18,A -85,B 0,C 180,E1 -25849.224,E2 -25849.224} C_VEL
LIN {X 0,Y 112.132,Z 462.874,A -85,B 0,C 180,E1 -25856.022,E2 -25856.022} C_VEL
LIN {X 0,Y 112.921,Z 463.387,A -85,B 0,C 180,E1 -25859.86,E2 -25859.86} C_VEL
LIN {X 0,Y 115.809,Z 463.394,A -85,B 0,C 180,E1 -25867.913,E2 -25867.913} C_VEL
LIN {X 0,Y 119.952,Z 462.185,A -85,B 0,C 180,E1 -25874.673,E2 -25874.673} C_VEL
LIN {X 0,Y 125.899,Z 459.559,A -85,B 0,C 180,E1 -25881.398,E2 -25881.398} C_VEL
LIN {X 0,Y 133.368,Z 455.505,A -85,B 0,C 180,E1 -25887.471,E2 -25887.471} C_VEL
LIN {X 0,Y 142.139,Z 449.917,A -85,B 0,C 180,E1 -25892.872,E2 -25892.872} C_VEL
LIN {X 0,Y 149.447,Z 444.58,A -85,B 0,C 180,E1 -25896.492,E2 -25896.492} C_VEL
LIN {X 0,Y 158.682,Z 437.055,A -85,B 0,C 180,E1 -25900.244,E2 -25900.244} C_VEL
LIN {X 0,Y 168.531,Z 427.852,A -85,B 0,C 180,E1 -25903.561,E2 -25903.561} C_VEL
LIN {X 0,Y 177.903,Z 417.699,A -85,B 0,C 180,E1 -25906.288,E2 -25906.288} C_VEL
LIN {X 0,Y 186.521,Z 406.978,A -85,B 0,C 180,E1 -25908.422,E2 -25908.422} C_VEL
LIN {X 0,Y 195.157,Z 394.398,A -85,B 0,C 180,E1 -25910.339,E2 -25910.339} C_VEL
LIN {X 0,Y 202.084,Z 382.494,A -85,B 0,C 180,E1 -25911.746,E2 -25911.746} C_VEL
LIN {X 0,Y 208.055,Z 370.407,A -85,B 0,C 180,E1 -25912.869,E2 -25912.869} C_VEL
LIN {X 0,Y 213.379,Z 357.393,A -85,B 0,C 180,E1 -25913.807,E2 -25913.807} C_VEL
LIN {X 0,Y 217.71,Z 344.03,A -85,B 0,C 180,E1 -25914.547,E2 -25914.547} C_VEL
LIN {X 0,Y 221.514,Z 328.509,A -85,B 0,C 180,E1 -25915.153,E2 -25915.153} C_VEL
LIN {X 0,Y 223.975,Z 312.949,A -85,B 0,C 180,E1 -25915.58,E2 -25915.58} C_VEL
LIN {X 0,Y 226.358,Z 291.019,A -85,B 0,C 180,E1 -25916.092,E2 -25916.092} C_VEL
LIN {X 0,Y 224.234,Z 285.95,A -85,B 0,C 180,E1 -25919.249,E2 -25919.249} C_VEL
LIN {X 0,Y 223.338,Z 283.929,A -85,B 0,C 180,E1 -25921.01,E2 -25921.01} C_VEL
LIN {X 0,Y 222.241,Z 280.947,A -85,B 0,C 180,E1 -25924.04,E2 -25924.04} C_VEL
LIN {X 0,Y 221.323,Z 279.787,A -85,B 0,C 180,E1 -25929.135,E2 -25929.135} C_VEL
LIN {X 0,Y 222.205,Z 281.343,A -85,B 0,C 180,E1 -25934.656,E2 -25934.656} C_VEL
LIN {X 0,Y 223.501,Z 284.791,A -85,B 0,C 180,E1 -25938.105,E2 -25938.105} C_VEL
LIN {X 0,Y 225.192,Z 289.97,A -85,B 0,C 180,E1 -25941.194,E2 -25941.194} C_VEL
LIN {X 0,Y 226.163,Z 293.19,A -85,B 0,C 180,E1 -25942.653,E2 -25942.653} C_VEL
LIN {X 0,Y 222.542,Z 324.319,A -85,B 0,C 180,E1 -25943.394,E2 -25943.394} C_VEL
LIN {X 0,Y 219.4,Z 339.707,A -85,B 0,C 180,E1 -25943.871,E2 -25943.871} C_VEL
LIN {X 0,Y 215.214,Z 354.128,A -85,B 0,C 180,E1 -25944.457,E2 -25944.457} C_VEL
LIN {X 0,Y 209.805,Z 368.475,A -85,B 0,C 180,E1 -25945.253,E2 -25945.253} C_VEL
LIN {X 0,Y 203.734,Z 381.556,A -85,B 0,C 180,E1 -25946.248,E2 -25946.248} C_VEL
LIN {X 0,Y 196.28,Z 394.928,A -85,B 0,C 180,E1 -25947.602,E2 -25947.602} C_VEL
LIN {X 0,Y 188.54,Z 406.609,A -85,B 0,C 180,E1 -25949.12,E2 -25949.12} C_VEL
LIN {X 0,Y 180.417,Z 417.367,A -85,B 0,C 180,E1 -25951.021,E2 -25951.021} C_VEL
LIN {X 0,Y 172.129,Z 426.939,A -85,B 0,C 180,E1 -25953.176,E2 -25953.176} C_VEL
LIN {X 0,Y 162.795,Z 436.386,A -85,B 0,C 180,E1 -25955.959,E2 -25955.959} C_VEL
LIN {X 0,Y 153.89,Z 444.314,A -85,B 0,C 180,E1 -25959.072,E2 -25959.072} C_VEL
LIN {X 0,Y 144.436,Z 451.759,A -85,B 0,C 180,E1 -25963.126,E2 -25963.126} C_VEL
LIN {X 0,Y 136.065,Z 457.745,A -85,B 0,C 180,E1 -25967.82,E2 -25967.82} C_VEL
LIN {X 0,Y 128.585,Z 462.389,A -85,B 0,C 180,E1 -25973.044,E2 -25973.044} C_VEL
LIN {X 0,Y 122.332,Z 465.805,A -85,B 0,C 180,E1 -25978.867,E2 -25978.867} C_VEL
LIN {X 0,Y 117.492,Z 468.086,A -85,B 0,C 180,E1 -25985.248,E2 -25985.248} C_VEL
LIN {X 0,Y 114.2,Z 469.281,A -85,B 0,C 180,E1 -25992.08,E2 -25992.08} C_VEL
LIN {X 0,Y 112.972,Z 469.451,A -85,B 0,C 180,E1 -25996.51,E2 -25996.51} C_VEL
LIN {X 0,Y 111.816,Z 469.337,A -85,B 0,C 180,E1 -25999.459,E2 -25999.459} C_VEL
LIN {X 0,Y 108.649,Z 468.561,A -85,B 0,C 180,E1 -26004.321,E2 -26004.321} C_VEL
LIN {X 0,Y 105.401,Z 466.886,A -85,B 0,C 180,E1 -26010.462,E2 -26010.462} C_VEL
LIN {X 0,Y 105.077,Z 466.112,A -85,B 0,C 180,E1 -26012.599,E2 -26012.599} C_VEL
LIN {X 0,Y 105.15,Z 464.042,A -85,B 0,C 180,E1 -26017.684,E2 -26017.684} C_VEL
LIN {X 0,Y 106.178,Z 459.76,A -85,B 0,C 180,E1 -26025.355,E2 -26025.355} C_VEL
LIN {X 0,Y 108.665,Z 454.047,A -85,B 0,C 180,E1 -26032.835,E2 -26032.835} C_VEL
LIN {X 0,Y 112.766,Z 446.758,A -85,B 0,C 180,E1 -26039.908,E2 -26039.908} C_VEL
LIN {X 0,Y 117.516,Z 438.913,A -85,B 0,C 180,E1 -26045.671,E2 -26045.671} C_VEL
LIN {X 0,Y 122.47,Z 430.942,A -85,B 0,C 180,E1 -26050.212,E2 -26050.212} C_VEL
LIN {X 0,Y 128.156,Z 421.223,A -85,B 0,C 180,E1 -26054.529,E2 -26054.529} C_VEL
LIN {X 0,Y 134.77,Z 409.286,A -85,B 0,C 180,E1 -26058.56,E2 -26058.56} C_VEL
LIN {X 0,Y 140.967,Z 396.809,A -85,B 0,C 180,E1 -26061.744,E2 -26061.744} C_VEL
LIN {X 0,Y 147.053,Z 383.083,A -85,B 0,C 180,E1 -26064.34,E2 -26064.34} C_VEL
LIN {X 0,Y 152.191,Z 369.152,A -85,B 0,C 180,E1 -26066.349,E2 -26066.349} C_VEL
LIN {X 0,Y 156.539,Z 354.868,A -85,B 0,C 180,E1 -26067.873,E2 -26067.873} C_VEL
LIN {X 0,Y 160.078,Z 339.827,A -85,B 0,C 180,E1 -26069.038,E2 -26069.038} C_VEL
LIN {X 0,Y 162.584,Z 324.75,A -85,B 0,C 180,E1 -26069.832,E2 -26069.832} C_VEL
LIN {X 0,Y 167.537,Z 270.989,A -85,B 0,C 180,E1 -26071.616,E2 -26071.616} C_VEL
LIN {X 0,Y 168.57,Z 258.956,A -85,B 0,C 180,E1 -26072.018,E2 -26072.018} C_VEL
LIN {X 0,Y 164.537,Z 246.811,A -85,B 0,C 180,E1 -26074.969,E2 -26074.969} C_VEL
LIN {X 0,Y 162.344,Z 241.29,A -85,B 0,C 180,E1 -26076.649,E2 -26076.649} C_VEL
LIN {X 0,Y 157.54,Z 232.337,A -85,B 0,C 180,E1 -26080.417,E2 -26080.417} C_VEL
LIN {X 0,Y 153.138,Z 225.011,A -85,B 0,C 180,E1 -26084.479,E2 -26084.479} C_VEL
LIN {X 0,Y 150.565,Z 220.866,A -85,B 0,C 180,E1 -26087.294,E2 -26087.294} C_VEL
LIN {X 0,Y 148.658,Z 217.762,A -85,B 0,C 180,E1 -26089.713,E2 -26089.713} C_VEL
LIN {X 0,Y 146.375,Z 214.273,A -85,B 0,C 180,E1 -26093.104,E2 -26093.104} C_VEL
LIN {X 0,Y 145.753,Z 213.314,A -85,B 0,C 180,E1 -26094.142,E2 -26094.142} C_VEL
LIN {X 0,Y 143.505,Z 210.024,A -85,B 0,C 180,E1 -26098.746,E2 -26098.746} C_VEL
LIN {X 0,Y 142.986,Z 208.634,A -85,B 0,C 180,E1 -26100.353,E2 -26100.353} C_VEL
LIN {X 0,Y 141.338,Z 207.687,A -85,B 0,C 180,E1 -26108.58,E2 -26108.58} C_VEL
LIN {X 0,Y 142.296,Z 208.803,A -85,B 0,C 180,E1 -26117.239,E2 -26117.239} C_VEL
LIN {X 0,Y 142.931,Z 209.282,A -85,B 0,C 180,E1 -26119.199,E2 -26119.199} C_VEL
LIN {X 0,Y 144.72,Z 212.657,A -85,B 0,C 180,E1 -26123.625,E2 -26123.625} C_VEL
LIN {X 0,Y 146.205,Z 214.266,A -85,B 0,C 180,E1 -26126.154,E2 -26126.154} C_VEL
LIN {X 0,Y 148.694,Z 218.031,A -85,B 0,C 180,E1 -26129.839,E2 -26129.839} C_VEL
LIN {X 0,Y 151.908,Z 223.2,A -85,B 0,C 180,E1 -26133.724,E2 -26133.724} C_VEL
LIN {X 0,Y 155.331,Z 228.624,A -85,B 0,C 180,E1 -26137.12,E2 -26137.12} C_VEL
LIN {X 0,Y 160.295,Z 237.46,A -85,B 0,C 180,E1 -26141.302,E2 -26141.302} C_VEL
LIN {X 0,Y 164.338,Z 245.415,A -85,B 0,C 180,E1 -26144.284,E2 -26144.284} C_VEL
LIN {X 0,Y 168.735,Z 255.234,A -85,B 0,C 180,E1 -26147.258,E2 -26147.258} C_VEL
